   1:  PR[GP1:91,1] = PR[GP1:90,1] + 51.280;
   1:  PR[GP1:91,2] = PR[GP1:90,2] + -7.015;
   1:L PR[91] 10mm/sec CNT100;
   1:  PR[GP1:91,1] = PR[GP1:90,1] + 52.296;
   1:  PR[GP1:91,2] = PR[GP1:90,2] + 0.271;
   1:L PR[91] 10mm/sec CNT100;
   1:  PR[GP1:91,1] = PR[GP1:90,1] + 51.315;
   1:  PR[GP1:91,2] = PR[GP1:90,2] + 6.204;
   1:L PR[91] 10mm/sec CNT100;
   1:  PR[GP1:91,1] = PR[GP1:90,1] + 50.273;
   1:  PR[GP1:91,2] = PR[GP1:90,2] + 13.672;
   1:L PR[91] 10mm/sec CNT100;
   1:  PR[GP1:91,1] = PR[GP1:90,1] + 47.241;
   1:  PR[GP1:91,2] = PR[GP1:90,2] + 20.539;
   1:L PR[91] 10mm/sec CNT100;
   1:  PR[GP1:91,1] = PR[GP1:90,1] + 44.357;
   1:  PR[GP1:91,2] = PR[GP1:90,2] + 25.832;
   1:L PR[91] 10mm/sec CNT100;
   1:  PR[GP1:91,1] = PR[GP1:90,1] + 39.468;
   1:  PR[GP1:91,2] = PR[GP1:90,2] + 31.722;
   1:L PR[91] 10mm/sec CNT100;
   1:  PR[GP1:91,1] = PR[GP1:90,1] + 35.135;
   1:  PR[GP1:91,2] = PR[GP1:90,2] + 35.737;
   1:L PR[91] 10mm/sec CNT100;
   1:  PR[GP1:91,1] = PR[GP1:90,1] + 26.217;
   1:  PR[GP1:91,2] = PR[GP1:90,2] + 41.260;
   1:L PR[91] 10mm/sec CNT100;
   1:  PR[GP1:91,1] = PR[GP1:90,1] + 20.960;
   1:  PR[GP1:91,2] = PR[GP1:90,2] + 43.644;
   1:L PR[91] 10mm/sec CNT100;
   1:  PR[GP1:91,1] = PR[GP1:90,1] + 10.344;
   1:  PR[GP1:91,2] = PR[GP1:90,2] + 45.629;
   1:L PR[91] 10mm/sec CNT100;
   1:  PR[GP1:91,1] = PR[GP1:90,1] + 4.776;
   1:  PR[GP1:91,2] = PR[GP1:90,2] + 46.223;
   1:L PR[91] 10mm/sec CNT100;
   1:  PR[GP1:91,1] = PR[GP1:90,1] + -0.263;
   1:  PR[GP1:91,2] = PR[GP1:90,2] + 45.337;
   1:L PR[91] 10mm/sec CNT100;
   1:  PR[GP1:91,1] = PR[GP1:90,1] + -5.307;
   1:  PR[GP1:91,2] = PR[GP1:90,2] + 46.223;
   1:L PR[91] 10mm/sec CNT100;
   1:  PR[GP1:91,1] = PR[GP1:90,1] + -10.875;
   1:  PR[GP1:91,2] = PR[GP1:90,2] + 45.629;
   1:L PR[91] 10mm/sec CNT100;
   1:  PR[GP1:91,1] = PR[GP1:90,1] + -21.488;
   1:  PR[GP1:91,2] = PR[GP1:90,2] + 43.644;
   1:L PR[91] 10mm/sec CNT100;
   1:  PR[GP1:91,1] = PR[GP1:90,1] + -26.745;
   1:  PR[GP1:91,2] = PR[GP1:90,2] + 41.258;
   1:L PR[91] 10mm/sec CNT100;
   1:  PR[GP1:91,1] = PR[GP1:90,1] + -35.660;
   1:  PR[GP1:91,2] = PR[GP1:90,2] + 35.736;
   1:L PR[91] 10mm/sec CNT100;
   1:  PR[GP1:91,1] = PR[GP1:90,1] + -39.993;
   1:  PR[GP1:91,2] = PR[GP1:90,2] + 31.727;
   1:L PR[91] 10mm/sec CNT100;
   1:  PR[GP1:91,1] = PR[GP1:90,1] + -44.883;
   1:  PR[GP1:91,2] = PR[GP1:90,2] + 25.837;
   1:L PR[91] 10mm/sec CNT100;
   1:  PR[GP1:91,1] = PR[GP1:90,1] + -47.767;
   1:  PR[GP1:91,2] = PR[GP1:90,2] + 20.534;
   1:L PR[91] 10mm/sec CNT100;
   1:  PR[GP1:91,1] = PR[GP1:90,1] + -50.803;
   1:  PR[GP1:91,2] = PR[GP1:90,2] + 13.658;
   1:L PR[91] 10mm/sec CNT100;
   1:  PR[GP1:91,1] = PR[GP1:90,1] + -51.805;
   1:  PR[GP1:91,2] = PR[GP1:90,2] + 7.716;
   1:L PR[91] 10mm/sec CNT100;
   1:  PR[GP1:91,1] = PR[GP1:90,1] + -51.806;
   1:  PR[GP1:91,2] = PR[GP1:90,2] + 7.573;
   1:L PR[91] 10mm/sec CNT100;
   1:  PR[GP1:91,1] = PR[GP1:90,1] + -52.823;
   1:  PR[GP1:91,2] = PR[GP1:90,2] + 0.287;
   1:L PR[91] 10mm/sec CNT100;
   1:  PR[GP1:91,1] = PR[GP1:90,1] + -51.845;
   1:  PR[GP1:91,2] = PR[GP1:90,2] + -5.627;
   1:L PR[91] 10mm/sec CNT100;
   1:  PR[GP1:91,1] = PR[GP1:90,1] + -50.804;
   1:  PR[GP1:91,2] = PR[GP1:90,2] + -13.095;
   1:L PR[91] 10mm/sec CNT100;
   1:  PR[GP1:91,1] = PR[GP1:90,1] + -47.772;
   1:  PR[GP1:91,2] = PR[GP1:90,2] + -19.963;
   1:L PR[91] 10mm/sec CNT100;
   1:  PR[GP1:91,1] = PR[GP1:90,1] + -44.899;
   1:  PR[GP1:91,2] = PR[GP1:90,2] + -25.258;
   1:L PR[91] 10mm/sec CNT100;
   1:  PR[GP1:91,1] = PR[GP1:90,1] + -40.009;
   1:  PR[GP1:91,2] = PR[GP1:90,2] + -31.148;
   1:L PR[91] 10mm/sec CNT100;
   1:  PR[GP1:91,1] = PR[GP1:90,1] + -35.691;
   1:  PR[GP1:91,2] = PR[GP1:90,2] + -35.157;
   1:L PR[91] 10mm/sec CNT100;
   1:  PR[GP1:91,1] = PR[GP1:90,1] + -26.777;
   1:  PR[GP1:91,2] = PR[GP1:90,2] + -40.678;
   1:L PR[91] 10mm/sec CNT100;
   1:  PR[GP1:91,1] = PR[GP1:90,1] + -21.535;
   1:  PR[GP1:91,2] = PR[GP1:90,2] + -43.073;
   1:L PR[91] 10mm/sec CNT100;
   1:  PR[GP1:91,1] = PR[GP1:90,1] + -10.924;
   1:  PR[GP1:91,2] = PR[GP1:90,2] + -45.058;
   1:L PR[91] 10mm/sec CNT100;
   1:  PR[GP1:91,1] = PR[GP1:90,1] + -5.362;
   1:  PR[GP1:91,2] = PR[GP1:90,2] + -45.668;
   1:L PR[91] 10mm/sec CNT100;
   1:  PR[GP1:91,1] = PR[GP1:90,1] + -0.263;
   1:  PR[GP1:91,2] = PR[GP1:90,2] + -44.813;
   1:L PR[91] 10mm/sec CNT100;
   1:  PR[GP1:91,1] = PR[GP1:90,1] + 4.642;
   1:  PR[GP1:91,2] = PR[GP1:90,2] + -45.797;
   1:  PR[GP1:91,3] = PR[GP1:90,3] + 112.545;
   1:L PR[91] 10mm/sec CNT100;
   1:  PR[GP1:91,1] = PR[GP1:90,1] + 9.992;
   1:  PR[GP1:91,2] = PR[GP1:90,2] + -45.209;
   1:L PR[91] 10mm/sec CNT100;
   1:  PR[GP1:91,1] = PR[GP1:90,1] + 20.880;
   1:  PR[GP1:91,2] = PR[GP1:90,2] + -43.174;
   1:L PR[91] 10mm/sec CNT100;
   1:  PR[GP1:91,1] = PR[GP1:90,1] + 25.924;
   1:  PR[GP1:91,2] = PR[GP1:90,2] + -40.872;
   1:L PR[91] 10mm/sec CNT100;
   1:  PR[GP1:91,1] = PR[GP1:90,1] + 35.087;
   1:  PR[GP1:91,2] = PR[GP1:90,2] + -35.196;
   1:L PR[91] 10mm/sec CNT100;
   1:  PR[GP1:91,1] = PR[GP1:90,1] + 39.242;
   1:  PR[GP1:91,2] = PR[GP1:90,2] + -31.334;
   1:L PR[91] 10mm/sec CNT100;
   1:  PR[GP1:91,1] = PR[GP1:90,1] + 44.275;
   1:  PR[GP1:91,2] = PR[GP1:90,2] + -25.271;
   1:L PR[91] 10mm/sec CNT100;
   1:  PR[GP1:91,1] = PR[GP1:90,1] + 47.039;
   1:  PR[GP1:91,2] = PR[GP1:90,2] + -20.185;
   1:L PR[91] 10mm/sec CNT100;
   1:  PR[GP1:91,1] = PR[GP1:90,1] + 50.168;
   1:  PR[GP1:91,2] = PR[GP1:90,2] + -13.099;
   1:L PR[91] 10mm/sec CNT100;
   1:  PR[GP1:91,1] = PR[GP1:90,1] + 51.128;
   1:  PR[GP1:91,2] = PR[GP1:90,2] + -7.389;
   1:L PR[91] 10mm/sec CNT100;
   1:  PR[GP1:91,1] = PR[GP1:90,1] + 51.129;
   1:  PR[GP1:91,2] = PR[GP1:90,2] + -7.251;
   1:L PR[91] 10mm/sec CNT100;
   1:  PR[GP1:91,1] = PR[GP1:90,1] + 52.178;
   1:  PR[GP1:91,2] = PR[GP1:90,2] + 0.271;
   1:L PR[91] 10mm/sec CNT100;
   1:  PR[GP1:91,1] = PR[GP1:90,1] + 51.234;
   1:  PR[GP1:91,2] = PR[GP1:90,2] + 5.979;
   1:L PR[91] 10mm/sec CNT100;
   1:  PR[GP1:91,1] = PR[GP1:90,1] + 50.160;
   1:  PR[GP1:91,2] = PR[GP1:90,2] + 13.676;
   1:L PR[91] 10mm/sec CNT100;
   1:  PR[GP1:91,1] = PR[GP1:90,1] + 47.035;
   1:  PR[GP1:91,2] = PR[GP1:90,2] + 20.755;
   1:L PR[91] 10mm/sec CNT100;
   1:  PR[GP1:91,1] = PR[GP1:90,1] + 44.260;
   1:  PR[GP1:91,2] = PR[GP1:90,2] + 25.848;
   1:L PR[91] 10mm/sec CNT100;
   1:  PR[GP1:91,1] = PR[GP1:90,1] + 39.227;
   1:  PR[GP1:91,2] = PR[GP1:90,2] + 31.912;
   1:L PR[91] 10mm/sec CNT100;
   1:  PR[GP1:91,1] = PR[GP1:90,1] + 35.058;
   1:  PR[GP1:91,2] = PR[GP1:90,2] + 35.774;
   1:L PR[91] 10mm/sec CNT100;
   1:  PR[GP1:91,1] = PR[GP1:90,1] + 25.893;
   1:  PR[GP1:91,2] = PR[GP1:90,2] + 41.450;
   1:L PR[91] 10mm/sec CNT100;
   1:  PR[GP1:91,1] = PR[GP1:90,1] + 20.836;
   1:  PR[GP1:91,2] = PR[GP1:90,2] + 43.744;
   1:L PR[91] 10mm/sec CNT100;
   1:  PR[GP1:91,1] = PR[GP1:90,1] + 9.945;
   1:  PR[GP1:91,2] = PR[GP1:90,2] + 45.780;
   1:L PR[91] 10mm/sec CNT100;
   1:  PR[GP1:91,1] = PR[GP1:90,1] + 4.588;
   1:  PR[GP1:91,2] = PR[GP1:90,2] + 46.352;
   1:L PR[91] 10mm/sec CNT100;
   1:  PR[GP1:91,1] = PR[GP1:90,1] + -0.263;
   1:  PR[GP1:91,2] = PR[GP1:90,2] + 45.499;
   1:L PR[91] 10mm/sec CNT100;
   1:  PR[GP1:91,1] = PR[GP1:90,1] + -5.120;
   1:  PR[GP1:91,2] = PR[GP1:90,2] + 46.352;
   1:L PR[91] 10mm/sec CNT100;
   1:  PR[GP1:91,1] = PR[GP1:90,1] + -10.477;
   1:  PR[GP1:91,2] = PR[GP1:90,2] + 45.780;
   1:L PR[91] 10mm/sec CNT100;
   1:  PR[GP1:91,1] = PR[GP1:90,1] + -21.364;
   1:  PR[GP1:91,2] = PR[GP1:90,2] + 43.744;
   1:L PR[91] 10mm/sec CNT100;
   1:  PR[GP1:91,1] = PR[GP1:90,1] + -26.421;
   1:  PR[GP1:91,2] = PR[GP1:90,2] + 41.448;
   1:L PR[91] 10mm/sec CNT100;
   1:  PR[GP1:91,1] = PR[GP1:90,1] + -35.583;
   1:  PR[GP1:91,2] = PR[GP1:90,2] + 35.774;
   1:L PR[91] 10mm/sec CNT100;
   1:  PR[GP1:91,1] = PR[GP1:90,1] + -39.752;
   1:  PR[GP1:91,2] = PR[GP1:90,2] + 31.916;
   1:L PR[91] 10mm/sec CNT100;
   1:  PR[GP1:91,1] = PR[GP1:90,1] + -44.786;
   1:  PR[GP1:91,2] = PR[GP1:90,2] + 25.852;
   1:L PR[91] 10mm/sec CNT100;
   1:  PR[GP1:91,1] = PR[GP1:90,1] + -47.561;
   1:  PR[GP1:91,2] = PR[GP1:90,2] + 20.750;
   1:L PR[91] 10mm/sec CNT100;
   1:  PR[GP1:91,1] = PR[GP1:90,1] + -50.690;
   1:  PR[GP1:91,2] = PR[GP1:90,2] + 13.662;
   1:L PR[91] 10mm/sec CNT100;
   1:  PR[GP1:91,1] = PR[GP1:90,1] + -51.654;
   1:  PR[GP1:91,2] = PR[GP1:90,2] + 7.947;
   1:L PR[91] 10mm/sec CNT100;
   1:  PR[GP1:91,1] = PR[GP1:90,1] + -51.655;
   1:  PR[GP1:91,2] = PR[GP1:90,2] + 7.809;
   1:L PR[91] 10mm/sec CNT100;
   1:  PR[GP1:91,1] = PR[GP1:90,1] + -52.705;
   1:  PR[GP1:91,2] = PR[GP1:90,2] + 0.287;
   1:L PR[91] 10mm/sec CNT100;
   1:  PR[GP1:91,1] = PR[GP1:90,1] + -51.764;
   1:  PR[GP1:91,2] = PR[GP1:90,2] + -5.404;
   1:L PR[91] 10mm/sec CNT100;
   1:  PR[GP1:91,1] = PR[GP1:90,1] + -50.691;
   1:  PR[GP1:91,2] = PR[GP1:90,2] + -13.100;
   1:L PR[91] 10mm/sec CNT100;
   1:  PR[GP1:91,1] = PR[GP1:90,1] + -47.565;
   1:  PR[GP1:91,2] = PR[GP1:90,2] + -20.180;
   1:L PR[91] 10mm/sec CNT100;
   1:  PR[GP1:91,1] = PR[GP1:90,1] + -44.801;
   1:  PR[GP1:91,2] = PR[GP1:90,2] + -25.275;
   1:L PR[91] 10mm/sec CNT100;
   1:  PR[GP1:91,1] = PR[GP1:90,1] + -39.767;
   1:  PR[GP1:91,2] = PR[GP1:90,2] + -31.338;
   1:L PR[91] 10mm/sec CNT100;
   1:  PR[GP1:91,1] = PR[GP1:90,1] + -35.613;
   1:  PR[GP1:91,2] = PR[GP1:90,2] + -35.196;
   1:L PR[91] 10mm/sec CNT100;
   1:  PR[GP1:91,1] = PR[GP1:90,1] + -26.452;
   1:  PR[GP1:91,2] = PR[GP1:90,2] + -40.870;
   1:L PR[91] 10mm/sec CNT100;
   1:  PR[GP1:91,1] = PR[GP1:90,1] + -21.409;
   1:  PR[GP1:91,2] = PR[GP1:90,2] + -43.174;
   1:L PR[91] 10mm/sec CNT100;
   1:  PR[GP1:91,1] = PR[GP1:90,1] + -10.524;
   1:  PR[GP1:91,2] = PR[GP1:90,2] + -45.210;
   1:L PR[91] 10mm/sec CNT100;
   1:  PR[GP1:91,1] = PR[GP1:90,1] + -5.173;
   1:  PR[GP1:91,2] = PR[GP1:90,2] + -45.797;
   1:L PR[91] 10mm/sec CNT100;
   1:  PR[GP1:91,1] = PR[GP1:90,1] + -0.263;
   1:  PR[GP1:91,2] = PR[GP1:90,2] + -44.973;
   1:L PR[91] 10mm/sec CNT100;
   1:  PR[GP1:91,1] = PR[GP1:90,1] + 4.452;
   1:  PR[GP1:91,2] = PR[GP1:90,2] + -45.925;
   1:  PR[GP1:91,3] = PR[GP1:90,3] + 113.155;
   1:L PR[91] 10mm/sec CNT100;
   1:  PR[GP1:91,1] = PR[GP1:90,1] + 9.591;
   1:  PR[GP1:91,2] = PR[GP1:90,2] + -45.361;
   1:L PR[91] 10mm/sec CNT100;
   1:  PR[GP1:91,1] = PR[GP1:90,1] + 20.754;
   1:  PR[GP1:91,2] = PR[GP1:90,2] + -43.274;
   1:L PR[91] 10mm/sec CNT100;
   1:  PR[GP1:91,1] = PR[GP1:90,1] + 25.598;
   1:  PR[GP1:91,2] = PR[GP1:90,2] + -41.063;
   1:L PR[91] 10mm/sec CNT100;
   1:  PR[GP1:91,1] = PR[GP1:90,1] + 35.009;
   1:  PR[GP1:91,2] = PR[GP1:90,2] + -35.235;
   1:L PR[91] 10mm/sec CNT100;
   1:  PR[GP1:91,1] = PR[GP1:90,1] + 39.000;
   1:  PR[GP1:91,2] = PR[GP1:90,2] + -31.525;
   1:L PR[91] 10mm/sec CNT100;
   1:  PR[GP1:91,1] = PR[GP1:90,1] + 44.178;
   1:  PR[GP1:91,2] = PR[GP1:90,2] + -25.287;
   1:L PR[91] 10mm/sec CNT100;
   1:  PR[GP1:91,1] = PR[GP1:90,1] + 46.833;
   1:  PR[GP1:91,2] = PR[GP1:90,2] + -20.402;
   1:L PR[91] 10mm/sec CNT100;
   1:  PR[GP1:91,1] = PR[GP1:90,1] + 50.055;
   1:  PR[GP1:91,2] = PR[GP1:90,2] + -13.104;
   1:L PR[91] 10mm/sec CNT100;
   1:  PR[GP1:91,1] = PR[GP1:90,1] + 50.977;
   1:  PR[GP1:91,2] = PR[GP1:90,2] + -7.619;
   1:L PR[91] 10mm/sec CNT100;
   1:  PR[GP1:91,1] = PR[GP1:90,1] + 50.978;
   1:  PR[GP1:91,2] = PR[GP1:90,2] + -7.487;
   1:L PR[91] 10mm/sec CNT100;
   1:  PR[GP1:91,1] = PR[GP1:90,1] + 52.060;
   1:  PR[GP1:91,2] = PR[GP1:90,2] + 0.271;
   1:L PR[91] 10mm/sec CNT100;
   1:  PR[GP1:91,1] = PR[GP1:90,1] + 51.153;
   1:  PR[GP1:91,2] = PR[GP1:90,2] + 5.755;
   1:L PR[91] 10mm/sec CNT100;
   1:  PR[GP1:91,1] = PR[GP1:90,1] + 50.048;
   1:  PR[GP1:91,2] = PR[GP1:90,2] + 13.681;
   1:L PR[91] 10mm/sec CNT100;
   1:  PR[GP1:91,1] = PR[GP1:90,1] + 46.829;
   1:  PR[GP1:91,2] = PR[GP1:90,2] + 20.971;
   1:L PR[91] 10mm/sec CNT100;
   1:  PR[GP1:91,1] = PR[GP1:90,1] + 44.163;
   1:  PR[GP1:91,2] = PR[GP1:90,2] + 25.864;
   1:L PR[91] 10mm/sec CNT100;
   1:  PR[GP1:91,1] = PR[GP1:90,1] + 38.985;
   1:  PR[GP1:91,2] = PR[GP1:90,2] + 32.102;
   1:L PR[91] 10mm/sec CNT100;
   1:  PR[GP1:91,1] = PR[GP1:90,1] + 34.980;
   1:  PR[GP1:91,2] = PR[GP1:90,2] + 35.812;
   1:L PR[91] 10mm/sec CNT100;
   1:  PR[GP1:91,1] = PR[GP1:90,1] + 25.569;
   1:  PR[GP1:91,2] = PR[GP1:90,2] + 41.641;
   1:L PR[91] 10mm/sec CNT100;
   1:  PR[GP1:91,1] = PR[GP1:90,1] + 20.711;
   1:  PR[GP1:91,2] = PR[GP1:90,2] + 43.844;
   1:L PR[91] 10mm/sec CNT100;
   1:  PR[GP1:91,1] = PR[GP1:90,1] + 9.547;
   1:  PR[GP1:91,2] = PR[GP1:90,2] + 45.931;
   1:L PR[91] 10mm/sec CNT100;
   1:  PR[GP1:91,1] = PR[GP1:90,1] + 4.401;
   1:  PR[GP1:91,2] = PR[GP1:90,2] + 46.480;
   1:L PR[91] 10mm/sec CNT100;
   1:  PR[GP1:91,1] = PR[GP1:90,1] + -0.263;
   1:  PR[GP1:91,2] = PR[GP1:90,2] + 45.660;
   1:L PR[91] 10mm/sec CNT100;
   1:  PR[GP1:91,1] = PR[GP1:90,1] + -4.933;
   1:  PR[GP1:91,2] = PR[GP1:90,2] + 46.480;
   1:L PR[91] 10mm/sec CNT100;
   1:  PR[GP1:91,1] = PR[GP1:90,1] + -10.078;
   1:  PR[GP1:91,2] = PR[GP1:90,2] + 45.931;
   1:L PR[91] 10mm/sec CNT100;
   1:  PR[GP1:91,1] = PR[GP1:90,1] + -21.240;
   1:  PR[GP1:91,2] = PR[GP1:90,2] + 43.844;
   1:L PR[91] 10mm/sec CNT100;
   1:  PR[GP1:91,1] = PR[GP1:90,1] + -26.097;
   1:  PR[GP1:91,2] = PR[GP1:90,2] + 41.639;
   1:L PR[91] 10mm/sec CNT100;
   1:  PR[GP1:91,1] = PR[GP1:90,1] + -35.506;
   1:  PR[GP1:91,2] = PR[GP1:90,2] + 35.811;
   1:L PR[91] 10mm/sec CNT100;
   1:  PR[GP1:91,1] = PR[GP1:90,1] + -39.511;
   1:  PR[GP1:91,2] = PR[GP1:90,2] + 32.106;
   1:L PR[91] 10mm/sec CNT100;
   1:  PR[GP1:91,1] = PR[GP1:90,1] + -44.689;
   1:  PR[GP1:91,2] = PR[GP1:90,2] + 25.868;
   1:L PR[91] 10mm/sec CNT100;
   1:  PR[GP1:91,1] = PR[GP1:90,1] + -47.355;
   1:  PR[GP1:91,2] = PR[GP1:90,2] + 20.966;
   1:L PR[91] 10mm/sec CNT100;
   1:  PR[GP1:91,1] = PR[GP1:90,1] + -50.577;
   1:  PR[GP1:91,2] = PR[GP1:90,2] + 13.667;
   1:L PR[91] 10mm/sec CNT100;
   1:  PR[GP1:91,1] = PR[GP1:90,1] + -51.503;
   1:  PR[GP1:91,2] = PR[GP1:90,2] + 8.177;
   1:L PR[91] 10mm/sec CNT100;
   1:  PR[GP1:91,1] = PR[GP1:90,1] + -51.504;
   1:  PR[GP1:91,2] = PR[GP1:90,2] + 8.046;
   1:L PR[91] 10mm/sec CNT100;
   1:  PR[GP1:91,1] = PR[GP1:90,1] + -52.587;
   1:  PR[GP1:91,2] = PR[GP1:90,2] + 0.287;
   1:L PR[91] 10mm/sec CNT100;
   1:  PR[GP1:91,1] = PR[GP1:90,1] + -51.683;
   1:  PR[GP1:91,2] = PR[GP1:90,2] + -5.180;
   1:L PR[91] 10mm/sec CNT100;
   1:  PR[GP1:91,1] = PR[GP1:90,1] + -50.578;
   1:  PR[GP1:91,2] = PR[GP1:90,2] + -13.106;
   1:L PR[91] 10mm/sec CNT100;
   1:  PR[GP1:91,1] = PR[GP1:90,1] + -47.359;
   1:  PR[GP1:91,2] = PR[GP1:90,2] + -20.396;
   1:L PR[91] 10mm/sec CNT100;
   1:  PR[GP1:91,1] = PR[GP1:90,1] + -44.704;
   1:  PR[GP1:91,2] = PR[GP1:90,2] + -25.291;
   1:L PR[91] 10mm/sec CNT100;
   1:  PR[GP1:91,1] = PR[GP1:90,1] + -39.525;
   1:  PR[GP1:91,2] = PR[GP1:90,2] + -31.529;
   1:L PR[91] 10mm/sec CNT100;
   1:  PR[GP1:91,1] = PR[GP1:90,1] + -35.535;
   1:  PR[GP1:91,2] = PR[GP1:90,2] + -35.234;
   1:L PR[91] 10mm/sec CNT100;
   1:  PR[GP1:91,1] = PR[GP1:90,1] + -26.127;
   1:  PR[GP1:91,2] = PR[GP1:90,2] + -41.061;
   1:L PR[91] 10mm/sec CNT100;
   1:  PR[GP1:91,1] = PR[GP1:90,1] + -21.282;
   1:  PR[GP1:91,2] = PR[GP1:90,2] + -43.274;
   1:L PR[91] 10mm/sec CNT100;
   1:  PR[GP1:91,1] = PR[GP1:90,1] + -10.123;
   1:  PR[GP1:91,2] = PR[GP1:90,2] + -45.361;
   1:L PR[91] 10mm/sec CNT100;
   1:  PR[GP1:91,1] = PR[GP1:90,1] + -4.984;
   1:  PR[GP1:91,2] = PR[GP1:90,2] + -45.925;
   1:L PR[91] 10mm/sec CNT100;
   1:  PR[GP1:91,1] = PR[GP1:90,1] + -0.263;
   1:  PR[GP1:91,2] = PR[GP1:90,2] + -45.134;
   1:L PR[91] 10mm/sec CNT100;
   1:  PR[GP1:91,1] = PR[GP1:90,1] + 4.263;
   1:  PR[GP1:91,2] = PR[GP1:90,2] + -46.054;
   1:  PR[GP1:91,3] = PR[GP1:90,3] + 113.765;
   1:L PR[91] 10mm/sec CNT100;
   1:  PR[GP1:91,1] = PR[GP1:90,1] + 9.191;
   1:  PR[GP1:91,2] = PR[GP1:90,2] + -45.512;
   1:L PR[91] 10mm/sec CNT100;
   1:  PR[GP1:91,1] = PR[GP1:90,1] + 20.628;
   1:  PR[GP1:91,2] = PR[GP1:90,2] + -43.375;
   1:L PR[91] 10mm/sec CNT100;
   1:  PR[GP1:91,1] = PR[GP1:90,1] + 25.273;
   1:  PR[GP1:91,2] = PR[GP1:90,2] + -41.254;
   1:L PR[91] 10mm/sec CNT100;
   1:  PR[GP1:91,1] = PR[GP1:90,1] + 34.931;
   1:  PR[GP1:91,2] = PR[GP1:90,2] + -35.273;
   1:L PR[91] 10mm/sec CNT100;
   1:  PR[GP1:91,1] = PR[GP1:90,1] + 38.758;
   1:  PR[GP1:91,2] = PR[GP1:90,2] + -31.715;
   1:L PR[91] 10mm/sec CNT100;
   1:  PR[GP1:91,1] = PR[GP1:90,1] + 44.080;
   1:  PR[GP1:91,2] = PR[GP1:90,2] + -25.304;
   1:L PR[91] 10mm/sec CNT100;
   1:  PR[GP1:91,1] = PR[GP1:90,1] + 46.627;
   1:  PR[GP1:91,2] = PR[GP1:90,2] + -20.618;
   1:L PR[91] 10mm/sec CNT100;
   1:  PR[GP1:91,1] = PR[GP1:90,1] + 49.942;
   1:  PR[GP1:91,2] = PR[GP1:90,2] + -13.109;
   1:L PR[91] 10mm/sec CNT100;
   1:  PR[GP1:91,1] = PR[GP1:90,1] + 50.826;
   1:  PR[GP1:91,2] = PR[GP1:90,2] + -7.850;
   1:L PR[91] 10mm/sec CNT100;
   1:  PR[GP1:91,1] = PR[GP1:90,1] + 50.827;
   1:  PR[GP1:91,2] = PR[GP1:90,2] + -7.724;
   1:L PR[91] 10mm/sec CNT100;
   1:  PR[GP1:91,1] = PR[GP1:90,1] + 51.942;
   1:  PR[GP1:91,2] = PR[GP1:90,2] + 0.271;
   1:L PR[91] 10mm/sec CNT100;
   1:  PR[GP1:91,1] = PR[GP1:90,1] + 51.072;
   1:  PR[GP1:91,2] = PR[GP1:90,2] + 5.531;
   1:L PR[91] 10mm/sec CNT100;
   1:  PR[GP1:91,1] = PR[GP1:90,1] + 49.935;
   1:  PR[GP1:91,2] = PR[GP1:90,2] + 13.685;
   1:L PR[91] 10mm/sec CNT100;
   1:  PR[GP1:91,1] = PR[GP1:90,1] + 46.623;
   1:  PR[GP1:91,2] = PR[GP1:90,2] + 21.187;
   1:L PR[91] 10mm/sec CNT100;
   1:  PR[GP1:91,1] = PR[GP1:90,1] + 44.066;
   1:  PR[GP1:91,2] = PR[GP1:90,2] + 25.880;
   1:L PR[91] 10mm/sec CNT100;
   1:  PR[GP1:91,1] = PR[GP1:90,1] + 38.744;
   1:  PR[GP1:91,2] = PR[GP1:90,2] + 32.291;
   1:L PR[91] 10mm/sec CNT100;
   1:  PR[GP1:91,1] = PR[GP1:90,1] + 34.903;
   1:  PR[GP1:91,2] = PR[GP1:90,2] + 35.849;
   1:L PR[91] 10mm/sec CNT100;
   1:  PR[GP1:91,1] = PR[GP1:90,1] + 25.244;
   1:  PR[GP1:91,2] = PR[GP1:90,2] + 41.831;
   1:L PR[91] 10mm/sec CNT100;
   1:  PR[GP1:91,1] = PR[GP1:90,1] + 20.587;
   1:  PR[GP1:91,2] = PR[GP1:90,2] + 43.944;
   1:L PR[91] 10mm/sec CNT100;
   1:  PR[GP1:91,1] = PR[GP1:90,1] + 9.148;
   1:  PR[GP1:91,2] = PR[GP1:90,2] + 46.082;
   1:L PR[91] 10mm/sec CNT100;
   1:  PR[GP1:91,1] = PR[GP1:90,1] + 4.214;
   1:  PR[GP1:91,2] = PR[GP1:90,2] + 46.609;
   1:L PR[91] 10mm/sec CNT100;
   1:  PR[GP1:91,1] = PR[GP1:90,1] + -0.263;
   1:  PR[GP1:91,2] = PR[GP1:90,2] + 45.821;
   1:L PR[91] 10mm/sec CNT100;
   1:  PR[GP1:91,1] = PR[GP1:90,1] + -4.746;
   1:  PR[GP1:91,2] = PR[GP1:90,2] + 46.609;
   1:L PR[91] 10mm/sec CNT100;
   1:  PR[GP1:91,1] = PR[GP1:90,1] + -9.679;
   1:  PR[GP1:91,2] = PR[GP1:90,2] + 46.082;
   1:L PR[91] 10mm/sec CNT100;
   1:  PR[GP1:91,1] = PR[GP1:90,1] + -21.115;
   1:  PR[GP1:91,2] = PR[GP1:90,2] + 43.944;
   1:L PR[91] 10mm/sec CNT100;
   1:  PR[GP1:91,1] = PR[GP1:90,1] + -25.772;
   1:  PR[GP1:91,2] = PR[GP1:90,2] + 41.829;
   1:L PR[91] 10mm/sec CNT100;
   1:  PR[GP1:91,1] = PR[GP1:90,1] + -35.429;
   1:  PR[GP1:91,2] = PR[GP1:90,2] + 35.849;
   1:L PR[91] 10mm/sec CNT100;
   1:  PR[GP1:91,1] = PR[GP1:90,1] + -39.269;
   1:  PR[GP1:91,2] = PR[GP1:90,2] + 32.295;
   1:L PR[91] 10mm/sec CNT100;
   1:  PR[GP1:91,1] = PR[GP1:90,1] + -44.592;
   1:  PR[GP1:91,2] = PR[GP1:90,2] + 25.884;
   1:L PR[91] 10mm/sec CNT100;
   1:  PR[GP1:91,1] = PR[GP1:90,1] + -47.149;
   1:  PR[GP1:91,2] = PR[GP1:90,2] + 21.182;
   1:L PR[91] 10mm/sec CNT100;
   1:  PR[GP1:91,1] = PR[GP1:90,1] + -50.465;
   1:  PR[GP1:91,2] = PR[GP1:90,2] + 13.672;
   1:L PR[91] 10mm/sec CNT100;
   1:  PR[GP1:91,1] = PR[GP1:90,1] + -51.352;
   1:  PR[GP1:91,2] = PR[GP1:90,2] + 8.408;
   1:L PR[91] 10mm/sec CNT100;
   1:  PR[GP1:91,1] = PR[GP1:90,1] + -51.353;
   1:  PR[GP1:91,2] = PR[GP1:90,2] + 8.282;
   1:L PR[91] 10mm/sec CNT100;
   1:  PR[GP1:91,1] = PR[GP1:90,1] + -52.469;
   1:  PR[GP1:91,2] = PR[GP1:90,2] + 0.287;
   1:L PR[91] 10mm/sec CNT100;
   1:  PR[GP1:91,1] = PR[GP1:90,1] + -51.602;
   1:  PR[GP1:91,2] = PR[GP1:90,2] + -4.957;
   1:L PR[91] 10mm/sec CNT100;
   1:  PR[GP1:91,1] = PR[GP1:90,1] + -50.465;
   1:  PR[GP1:91,2] = PR[GP1:90,2] + -13.111;
   1:L PR[91] 10mm/sec CNT100;
   1:  PR[GP1:91,1] = PR[GP1:90,1] + -47.153;
   1:  PR[GP1:91,2] = PR[GP1:90,2] + -20.613;
   1:L PR[91] 10mm/sec CNT100;
   1:  PR[GP1:91,1] = PR[GP1:90,1] + -44.606;
   1:  PR[GP1:91,2] = PR[GP1:90,2] + -25.308;
   1:L PR[91] 10mm/sec CNT100;
   1:  PR[GP1:91,1] = PR[GP1:90,1] + -39.283;
   1:  PR[GP1:91,2] = PR[GP1:90,2] + -31.719;
   1:L PR[91] 10mm/sec CNT100;
   1:  PR[GP1:91,1] = PR[GP1:90,1] + -35.456;
   1:  PR[GP1:91,2] = PR[GP1:90,2] + -35.272;
   1:L PR[91] 10mm/sec CNT100;
   1:  PR[GP1:91,1] = PR[GP1:90,1] + -25.801;
   1:  PR[GP1:91,2] = PR[GP1:90,2] + -41.252;
   1:L PR[91] 10mm/sec CNT100;
   1:  PR[GP1:91,1] = PR[GP1:90,1] + -21.156;
   1:  PR[GP1:91,2] = PR[GP1:90,2] + -43.374;
   1:L PR[91] 10mm/sec CNT100;
   1:  PR[GP1:91,1] = PR[GP1:90,1] + -9.723;
   1:  PR[GP1:91,2] = PR[GP1:90,2] + -45.513;
   1:L PR[91] 10mm/sec CNT100;
   1:  PR[GP1:91,1] = PR[GP1:90,1] + -4.795;
   1:  PR[GP1:91,2] = PR[GP1:90,2] + -46.054;
   1:L PR[91] 10mm/sec CNT100;
   1:  PR[GP1:91,1] = PR[GP1:90,1] + -0.263;
   1:  PR[GP1:91,2] = PR[GP1:90,2] + -45.294;
   1:L PR[91] 10mm/sec CNT100;
   1:  PR[GP1:91,1] = PR[GP1:90,1] + 4.074;
   1:  PR[GP1:91,2] = PR[GP1:90,2] + -46.182;
   1:  PR[GP1:91,3] = PR[GP1:90,3] + 114.375;
   1:L PR[91] 10mm/sec CNT100;
   1:  PR[GP1:91,1] = PR[GP1:90,1] + 8.790;
   1:  PR[GP1:91,2] = PR[GP1:90,2] + -45.664;
   1:L PR[91] 10mm/sec CNT100;
   1:  PR[GP1:91,1] = PR[GP1:90,1] + 20.502;
   1:  PR[GP1:91,2] = PR[GP1:90,2] + -43.475;
   1:L PR[91] 10mm/sec CNT100;
   1:  PR[GP1:91,1] = PR[GP1:90,1] + 24.948;
   1:  PR[GP1:91,2] = PR[GP1:90,2] + -41.446;
   1:L PR[91] 10mm/sec CNT100;
   1:  PR[GP1:91,1] = PR[GP1:90,1] + 34.852;
   1:  PR[GP1:91,2] = PR[GP1:90,2] + -35.311;
   1:L PR[91] 10mm/sec CNT100;
   1:  PR[GP1:91,1] = PR[GP1:90,1] + 38.516;
   1:  PR[GP1:91,2] = PR[GP1:90,2] + -31.905;
   1:L PR[91] 10mm/sec CNT100;
   1:  PR[GP1:91,1] = PR[GP1:90,1] + 43.982;
   1:  PR[GP1:91,2] = PR[GP1:90,2] + -25.321;
   1:L PR[91] 10mm/sec CNT100;
   1:  PR[GP1:91,1] = PR[GP1:90,1] + 46.421;
   1:  PR[GP1:91,2] = PR[GP1:90,2] + -20.834;
   1:L PR[91] 10mm/sec CNT100;
   1:  PR[GP1:91,1] = PR[GP1:90,1] + 49.829;
   1:  PR[GP1:91,2] = PR[GP1:90,2] + -13.114;
   1:L PR[91] 10mm/sec CNT100;
   1:  PR[GP1:91,1] = PR[GP1:90,1] + 50.675;
   1:  PR[GP1:91,2] = PR[GP1:90,2] + -8.081;
   1:L PR[91] 10mm/sec CNT100;
   1:  PR[GP1:91,1] = PR[GP1:90,1] + 50.676;
   1:  PR[GP1:91,2] = PR[GP1:90,2] + -7.960;
   1:L PR[91] 10mm/sec CNT100;
   1:  PR[GP1:91,1] = PR[GP1:90,1] + 51.824;
   1:  PR[GP1:91,2] = PR[GP1:90,2] + 0.271;
   1:L PR[91] 10mm/sec CNT100;
   1:  PR[GP1:91,1] = PR[GP1:90,1] + 50.991;
   1:  PR[GP1:91,2] = PR[GP1:90,2] + 5.307;
   1:L PR[91] 10mm/sec CNT100;
   1:  PR[GP1:91,1] = PR[GP1:90,1] + 49.822;
   1:  PR[GP1:91,2] = PR[GP1:90,2] + 13.690;
   1:L PR[91] 10mm/sec CNT100;
   1:  PR[GP1:91,1] = PR[GP1:90,1] + 46.417;
   1:  PR[GP1:91,2] = PR[GP1:90,2] + 21.403;
   1:L PR[91] 10mm/sec CNT100;
   1:  PR[GP1:91,1] = PR[GP1:90,1] + 43.969;
   1:  PR[GP1:91,2] = PR[GP1:90,2] + 25.896;
   1:L PR[91] 10mm/sec CNT100;
   1:  PR[GP1:91,1] = PR[GP1:90,1] + 38.503;
   1:  PR[GP1:91,2] = PR[GP1:90,2] + 32.481;
   1:L PR[91] 10mm/sec CNT100;
   1:  PR[GP1:91,1] = PR[GP1:90,1] + 34.826;
   1:  PR[GP1:91,2] = PR[GP1:90,2] + 35.887;
   1:L PR[91] 10mm/sec CNT100;
   1:  PR[GP1:91,1] = PR[GP1:90,1] + 24.920;
   1:  PR[GP1:91,2] = PR[GP1:90,2] + 42.022;
   1:L PR[91] 10mm/sec CNT100;
   1:  PR[GP1:91,1] = PR[GP1:90,1] + 20.462;
   1:  PR[GP1:91,2] = PR[GP1:90,2] + 44.044;
   1:L PR[91] 10mm/sec CNT100;
   1:  PR[GP1:91,1] = PR[GP1:90,1] + 8.749;
   1:  PR[GP1:91,2] = PR[GP1:90,2] + 46.233;
   1:L PR[91] 10mm/sec CNT100;
   1:  PR[GP1:91,1] = PR[GP1:90,1] + 4.027;
   1:  PR[GP1:91,2] = PR[GP1:90,2] + 46.737;
   1:L PR[91] 10mm/sec CNT100;
   1:  PR[GP1:91,1] = PR[GP1:90,1] + -0.263;
   1:  PR[GP1:91,2] = PR[GP1:90,2] + 45.983;
   1:L PR[91] 10mm/sec CNT100;
   1:  PR[GP1:91,1] = PR[GP1:90,1] + -4.559;
   1:  PR[GP1:91,2] = PR[GP1:90,2] + 46.737;
   1:L PR[91] 10mm/sec CNT100;
   1:  PR[GP1:91,1] = PR[GP1:90,1] + -9.281;
   1:  PR[GP1:91,2] = PR[GP1:90,2] + 46.234;
   1:L PR[91] 10mm/sec CNT100;
   1:  PR[GP1:91,1] = PR[GP1:90,1] + -20.991;
   1:  PR[GP1:91,2] = PR[GP1:90,2] + 44.043;
   1:L PR[91] 10mm/sec CNT100;
   1:  PR[GP1:91,1] = PR[GP1:90,1] + -25.448;
   1:  PR[GP1:91,2] = PR[GP1:90,2] + 42.020;
   1:L PR[91] 10mm/sec CNT100;
   1:  PR[GP1:91,1] = PR[GP1:90,1] + -35.352;
   1:  PR[GP1:91,2] = PR[GP1:90,2] + 35.886;
   1:L PR[91] 10mm/sec CNT100;
   1:  PR[GP1:91,1] = PR[GP1:90,1] + -39.028;
   1:  PR[GP1:91,2] = PR[GP1:90,2] + 32.485;
   1:L PR[91] 10mm/sec CNT100;
   1:  PR[GP1:91,1] = PR[GP1:90,1] + -44.495;
   1:  PR[GP1:91,2] = PR[GP1:90,2] + 25.899;
   1:L PR[91] 10mm/sec CNT100;
   1:  PR[GP1:91,1] = PR[GP1:90,1] + -46.943;
   1:  PR[GP1:91,2] = PR[GP1:90,2] + 21.398;
   1:L PR[91] 10mm/sec CNT100;
   1:  PR[GP1:91,1] = PR[GP1:90,1] + -50.352;
   1:  PR[GP1:91,2] = PR[GP1:90,2] + 13.677;
   1:L PR[91] 10mm/sec CNT100;
   1:  PR[GP1:91,1] = PR[GP1:90,1] + -51.201;
   1:  PR[GP1:91,2] = PR[GP1:90,2] + 8.639;
   1:L PR[91] 10mm/sec CNT100;
   1:  PR[GP1:91,1] = PR[GP1:90,1] + -51.203;
   1:  PR[GP1:91,2] = PR[GP1:90,2] + 8.518;
   1:L PR[91] 10mm/sec CNT100;
   1:  PR[GP1:91,1] = PR[GP1:90,1] + -52.351;
   1:  PR[GP1:91,2] = PR[GP1:90,2] + 0.287;
   1:L PR[91] 10mm/sec CNT100;
   1:  PR[GP1:91,1] = PR[GP1:90,1] + -51.521;
   1:  PR[GP1:91,2] = PR[GP1:90,2] + -4.733;
   1:L PR[91] 10mm/sec CNT100;
   1:  PR[GP1:91,1] = PR[GP1:90,1] + -50.352;
   1:  PR[GP1:91,2] = PR[GP1:90,2] + -13.116;
   1:L PR[91] 10mm/sec CNT100;
   1:  PR[GP1:91,1] = PR[GP1:90,1] + -46.947;
   1:  PR[GP1:91,2] = PR[GP1:90,2] + -20.830;
   1:L PR[91] 10mm/sec CNT100;
   1:  PR[GP1:91,1] = PR[GP1:90,1] + -44.508;
   1:  PR[GP1:91,2] = PR[GP1:90,2] + -25.324;
   1:L PR[91] 10mm/sec CNT100;
   1:  PR[GP1:91,1] = PR[GP1:90,1] + -39.042;
   1:  PR[GP1:91,2] = PR[GP1:90,2] + -31.909;
   1:L PR[91] 10mm/sec CNT100;
   1:  PR[GP1:91,1] = PR[GP1:90,1] + -35.378;
   1:  PR[GP1:91,2] = PR[GP1:90,2] + -35.311;
   1:L PR[91] 10mm/sec CNT100;
   1:  PR[GP1:91,1] = PR[GP1:90,1] + -25.476;
   1:  PR[GP1:91,2] = PR[GP1:90,2] + -41.444;
   1:L PR[91] 10mm/sec CNT100;
   1:  PR[GP1:91,1] = PR[GP1:90,1] + -21.030;
   1:  PR[GP1:91,2] = PR[GP1:90,2] + -43.475;
   1:L PR[91] 10mm/sec CNT100;
   1:  PR[GP1:91,1] = PR[GP1:90,1] + -9.322;
   1:  PR[GP1:91,2] = PR[GP1:90,2] + -45.664;
   1:L PR[91] 10mm/sec CNT100;
   1:  PR[GP1:91,1] = PR[GP1:90,1] + -4.605;
   1:  PR[GP1:91,2] = PR[GP1:90,2] + -46.182;
   1:L PR[91] 10mm/sec CNT100;
   1:  PR[GP1:91,1] = PR[GP1:90,1] + -0.263;
   1:  PR[GP1:91,2] = PR[GP1:90,2] + -45.454;
   1:L PR[91] 10mm/sec CNT100;
   1:  PR[GP1:91,1] = PR[GP1:90,1] + 3.884;
   1:  PR[GP1:91,2] = PR[GP1:90,2] + -46.311;
   1:  PR[GP1:91,3] = PR[GP1:90,3] + 114.985;
   1:L PR[91] 10mm/sec CNT100;
   1:  PR[GP1:91,1] = PR[GP1:90,1] + 8.390;
   1:  PR[GP1:91,2] = PR[GP1:90,2] + -45.816;
   1:L PR[91] 10mm/sec CNT100;
   1:  PR[GP1:91,1] = PR[GP1:90,1] + 20.375;
   1:  PR[GP1:91,2] = PR[GP1:90,2] + -43.575;
   1:L PR[91] 10mm/sec CNT100;
   1:  PR[GP1:91,1] = PR[GP1:90,1] + 24.622;
   1:  PR[GP1:91,2] = PR[GP1:90,2] + -41.637;
   1:L PR[91] 10mm/sec CNT100;
   1:  PR[GP1:91,1] = PR[GP1:90,1] + 34.774;
   1:  PR[GP1:91,2] = PR[GP1:90,2] + -35.350;
   1:L PR[91] 10mm/sec CNT100;
   1:  PR[GP1:91,1] = PR[GP1:90,1] + 38.274;
   1:  PR[GP1:91,2] = PR[GP1:90,2] + -32.096;
   1:L PR[91] 10mm/sec CNT100;
   1:  PR[GP1:91,1] = PR[GP1:90,1] + 43.885;
   1:  PR[GP1:91,2] = PR[GP1:90,2] + -25.337;
   1:L PR[91] 10mm/sec CNT100;
   1:  PR[GP1:91,1] = PR[GP1:90,1] + 46.215;
   1:  PR[GP1:91,2] = PR[GP1:90,2] + -21.050;
   1:L PR[91] 10mm/sec CNT100;
   1:  PR[GP1:91,1] = PR[GP1:90,1] + 49.716;
   1:  PR[GP1:91,2] = PR[GP1:90,2] + -13.119;
   1:L PR[91] 10mm/sec CNT100;
   1:  PR[GP1:91,1] = PR[GP1:90,1] + 50.524;
   1:  PR[GP1:91,2] = PR[GP1:90,2] + -8.311;
   1:L PR[91] 10mm/sec CNT100;
   1:  PR[GP1:91,1] = PR[GP1:90,1] + 50.525;
   1:  PR[GP1:91,2] = PR[GP1:90,2] + -8.196;
   1:L PR[91] 10mm/sec CNT100;
   1:  PR[GP1:91,1] = PR[GP1:90,1] + 51.706;
   1:  PR[GP1:91,2] = PR[GP1:90,2] + 0.271;
   1:L PR[91] 10mm/sec CNT100;
   1:  PR[GP1:91,1] = PR[GP1:90,1] + 50.910;
   1:  PR[GP1:91,2] = PR[GP1:90,2] + 5.083;
   1:L PR[91] 10mm/sec CNT100;
   1:  PR[GP1:91,1] = PR[GP1:90,1] + 49.709;
   1:  PR[GP1:91,2] = PR[GP1:90,2] + 13.694;
   1:L PR[91] 10mm/sec CNT100;
   1:  PR[GP1:91,1] = PR[GP1:90,1] + 46.211;
   1:  PR[GP1:91,2] = PR[GP1:90,2] + 21.618;
   1:L PR[91] 10mm/sec CNT100;
   1:  PR[GP1:91,1] = PR[GP1:90,1] + 43.872;
   1:  PR[GP1:91,2] = PR[GP1:90,2] + 25.912;
   1:L PR[91] 10mm/sec CNT100;
   1:  PR[GP1:91,1] = PR[GP1:90,1] + 38.261;
   1:  PR[GP1:91,2] = PR[GP1:90,2] + 32.670;
   1:L PR[91] 10mm/sec CNT100;
   1:  PR[GP1:91,1] = PR[GP1:90,1] + 34.749;
   1:  PR[GP1:91,2] = PR[GP1:90,2] + 35.924;
   1:L PR[91] 10mm/sec CNT100;
   1:  PR[GP1:91,1] = PR[GP1:90,1] + 24.596;
   1:  PR[GP1:91,2] = PR[GP1:90,2] + 42.212;
   1:L PR[91] 10mm/sec CNT100;
   1:  PR[GP1:91,1] = PR[GP1:90,1] + 20.338;
   1:  PR[GP1:91,2] = PR[GP1:90,2] + 44.144;
   1:L PR[91] 10mm/sec CNT100;
   1:  PR[GP1:91,1] = PR[GP1:90,1] + 8.351;
   1:  PR[GP1:91,2] = PR[GP1:90,2] + 46.384;
   1:L PR[91] 10mm/sec CNT100;
   1:  PR[GP1:91,1] = PR[GP1:90,1] + 3.840;
   1:  PR[GP1:91,2] = PR[GP1:90,2] + 46.866;
   1:L PR[91] 10mm/sec CNT100;
   1:  PR[GP1:91,1] = PR[GP1:90,1] + -0.264;
   1:  PR[GP1:91,2] = PR[GP1:90,2] + 46.144;
   1:L PR[91] 10mm/sec CNT100;
   1:  PR[GP1:91,1] = PR[GP1:90,1] + -4.372;
   1:  PR[GP1:91,2] = PR[GP1:90,2] + 46.866;
   1:L PR[91] 10mm/sec CNT100;
   1:  PR[GP1:91,1] = PR[GP1:90,1] + -8.882;
   1:  PR[GP1:91,2] = PR[GP1:90,2] + 46.385;
   1:L PR[91] 10mm/sec CNT100;
   1:  PR[GP1:91,1] = PR[GP1:90,1] + -20.866;
   1:  PR[GP1:91,2] = PR[GP1:90,2] + 44.143;
   1:L PR[91] 10mm/sec CNT100;
   1:  PR[GP1:91,1] = PR[GP1:90,1] + -25.124;
   1:  PR[GP1:91,2] = PR[GP1:90,2] + 42.210;
   1:L PR[91] 10mm/sec CNT100;
   1:  PR[GP1:91,1] = PR[GP1:90,1] + -35.274;
   1:  PR[GP1:91,2] = PR[GP1:90,2] + 35.924;
   1:L PR[91] 10mm/sec CNT100;
   1:  PR[GP1:91,1] = PR[GP1:90,1] + -38.787;
   1:  PR[GP1:91,2] = PR[GP1:90,2] + 32.674;
   1:L PR[91] 10mm/sec CNT100;
   1:  PR[GP1:91,1] = PR[GP1:90,1] + -44.398;
   1:  PR[GP1:91,2] = PR[GP1:90,2] + 25.915;
   1:L PR[91] 10mm/sec CNT100;
   1:  PR[GP1:91,1] = PR[GP1:90,1] + -46.737;
   1:  PR[GP1:91,2] = PR[GP1:90,2] + 21.614;
   1:L PR[91] 10mm/sec CNT100;
   1:  PR[GP1:91,1] = PR[GP1:90,1] + -50.239;
   1:  PR[GP1:91,2] = PR[GP1:90,2] + 13.682;
   1:L PR[91] 10mm/sec CNT100;
   1:  PR[GP1:91,1] = PR[GP1:90,1] + -51.050;
   1:  PR[GP1:91,2] = PR[GP1:90,2] + 8.870;
   1:L PR[91] 10mm/sec CNT100;
   1:  PR[GP1:91,1] = PR[GP1:90,1] + -51.052;
   1:  PR[GP1:91,2] = PR[GP1:90,2] + 8.755;
   1:L PR[91] 10mm/sec CNT100;
   1:  PR[GP1:91,1] = PR[GP1:90,1] + -52.233;
   1:  PR[GP1:91,2] = PR[GP1:90,2] + 0.287;
   1:L PR[91] 10mm/sec CNT100;
   1:  PR[GP1:91,1] = PR[GP1:90,1] + -51.440;
   1:  PR[GP1:91,2] = PR[GP1:90,2] + -4.510;
   1:L PR[91] 10mm/sec CNT100;
   1:  PR[GP1:91,1] = PR[GP1:90,1] + -50.239;
   1:  PR[GP1:91,2] = PR[GP1:90,2] + -13.122;
   1:L PR[91] 10mm/sec CNT100;
   1:  PR[GP1:91,1] = PR[GP1:90,1] + -46.740;
   1:  PR[GP1:91,2] = PR[GP1:90,2] + -21.046;
   1:L PR[91] 10mm/sec CNT100;
   1:  PR[GP1:91,1] = PR[GP1:90,1] + -44.411;
   1:  PR[GP1:91,2] = PR[GP1:90,2] + -25.341;
   1:L PR[91] 10mm/sec CNT100;
   1:  PR[GP1:91,1] = PR[GP1:90,1] + -38.800;
   1:  PR[GP1:91,2] = PR[GP1:90,2] + -32.099;
   1:L PR[91] 10mm/sec CNT100;
   1:  PR[GP1:91,1] = PR[GP1:90,1] + -35.299;
   1:  PR[GP1:91,2] = PR[GP1:90,2] + -35.349;
   1:L PR[91] 10mm/sec CNT100;
   1:  PR[GP1:91,1] = PR[GP1:90,1] + -25.151;
   1:  PR[GP1:91,2] = PR[GP1:90,2] + -41.635;
   1:L PR[91] 10mm/sec CNT100;
   1:  PR[GP1:91,1] = PR[GP1:90,1] + -20.904;
   1:  PR[GP1:91,2] = PR[GP1:90,2] + -43.575;
   1:L PR[91] 10mm/sec CNT100;
   1:  PR[GP1:91,1] = PR[GP1:90,1] + -8.922;
   1:  PR[GP1:91,2] = PR[GP1:90,2] + -45.816;
   1:L PR[91] 10mm/sec CNT100;
   1:  PR[GP1:91,1] = PR[GP1:90,1] + -4.416;
   1:  PR[GP1:91,2] = PR[GP1:90,2] + -46.311;
   1:L PR[91] 10mm/sec CNT100;
   1:  PR[GP1:91,1] = PR[GP1:90,1] + -0.264;
   1:  PR[GP1:91,2] = PR[GP1:90,2] + -45.614;
   1:L PR[91] 10mm/sec CNT100;
   1:  PR[GP1:91,1] = PR[GP1:90,1] + 3.695;
   1:  PR[GP1:91,2] = PR[GP1:90,2] + -46.439;
   1:  PR[GP1:91,3] = PR[GP1:90,3] + 115.595;
   1:L PR[91] 10mm/sec CNT100;
   1:  PR[GP1:91,1] = PR[GP1:90,1] + 7.989;
   1:  PR[GP1:91,2] = PR[GP1:90,2] + -45.967;
   1:L PR[91] 10mm/sec CNT100;
   1:  PR[GP1:91,1] = PR[GP1:90,1] + 20.249;
   1:  PR[GP1:91,2] = PR[GP1:90,2] + -43.676;
   1:L PR[91] 10mm/sec CNT100;
   1:  PR[GP1:91,1] = PR[GP1:90,1] + 24.297;
   1:  PR[GP1:91,2] = PR[GP1:90,2] + -41.828;
   1:L PR[91] 10mm/sec CNT100;
   1:  PR[GP1:91,1] = PR[GP1:90,1] + 34.695;
   1:  PR[GP1:91,2] = PR[GP1:90,2] + -35.388;
   1:L PR[91] 10mm/sec CNT100;
   1:  PR[GP1:91,1] = PR[GP1:90,1] + 38.032;
   1:  PR[GP1:91,2] = PR[GP1:90,2] + -32.286;
   1:L PR[91] 10mm/sec CNT100;
   1:  PR[GP1:91,1] = PR[GP1:90,1] + 43.787;
   1:  PR[GP1:91,2] = PR[GP1:90,2] + -25.354;
   1:L PR[91] 10mm/sec CNT100;
   1:  PR[GP1:91,1] = PR[GP1:90,1] + 46.008;
   1:  PR[GP1:91,2] = PR[GP1:90,2] + -21.267;
   1:L PR[91] 10mm/sec CNT100;
   1:  PR[GP1:91,1] = PR[GP1:90,1] + 49.603;
   1:  PR[GP1:91,2] = PR[GP1:90,2] + -13.124;
   1:L PR[91] 10mm/sec CNT100;
   1:  PR[GP1:91,1] = PR[GP1:90,1] + 50.373;
   1:  PR[GP1:91,2] = PR[GP1:90,2] + -8.542;
   1:L PR[91] 10mm/sec CNT100;
   1:  PR[GP1:91,1] = PR[GP1:90,1] + 50.374;
   1:  PR[GP1:91,2] = PR[GP1:90,2] + -8.433;
   1:L PR[91] 10mm/sec CNT100;
   1:  PR[GP1:91,1] = PR[GP1:90,1] + 51.588;
   1:  PR[GP1:91,2] = PR[GP1:90,2] + 0.271;
   1:L PR[91] 10mm/sec CNT100;
   1:  PR[GP1:91,1] = PR[GP1:90,1] + 50.829;
   1:  PR[GP1:91,2] = PR[GP1:90,2] + 4.859;
   1:L PR[91] 10mm/sec CNT100;
   1:  PR[GP1:91,1] = PR[GP1:90,1] + 49.596;
   1:  PR[GP1:91,2] = PR[GP1:90,2] + 13.699;
   1:L PR[91] 10mm/sec CNT100;
   1:  PR[GP1:91,1] = PR[GP1:90,1] + 46.005;
   1:  PR[GP1:91,2] = PR[GP1:90,2] + 21.834;
   1:L PR[91] 10mm/sec CNT100;
   1:  PR[GP1:91,1] = PR[GP1:90,1] + 43.775;
   1:  PR[GP1:91,2] = PR[GP1:90,2] + 25.928;
   1:L PR[91] 10mm/sec CNT100;
   1:  PR[GP1:91,1] = PR[GP1:90,1] + 38.020;
   1:  PR[GP1:91,2] = PR[GP1:90,2] + 32.860;
   1:L PR[91] 10mm/sec CNT100;
   1:  PR[GP1:91,1] = PR[GP1:90,1] + 34.672;
   1:  PR[GP1:91,2] = PR[GP1:90,2] + 35.962;
   1:L PR[91] 10mm/sec CNT100;
   1:  PR[GP1:91,1] = PR[GP1:90,1] + 24.272;
   1:  PR[GP1:91,2] = PR[GP1:90,2] + 42.403;
   1:L PR[91] 10mm/sec CNT100;
   1:  PR[GP1:91,1] = PR[GP1:90,1] + 20.213;
   1:  PR[GP1:91,2] = PR[GP1:90,2] + 44.244;
   1:L PR[91] 10mm/sec CNT100;
   1:  PR[GP1:91,1] = PR[GP1:90,1] + 7.952;
   1:  PR[GP1:91,2] = PR[GP1:90,2] + 46.535;
   1:L PR[91] 10mm/sec CNT100;
   1:  PR[GP1:91,1] = PR[GP1:90,1] + 3.653;
   1:  PR[GP1:91,2] = PR[GP1:90,2] + 46.995;
   1:L PR[91] 10mm/sec CNT100;
   1:  PR[GP1:91,1] = PR[GP1:90,1] + -0.264;
   1:  PR[GP1:91,2] = PR[GP1:90,2] + 46.306;
   1:L PR[91] 10mm/sec CNT100;
   1:  PR[GP1:91,1] = PR[GP1:90,1] + -4.185;
   1:  PR[GP1:91,2] = PR[GP1:90,2] + 46.994;
   1:L PR[91] 10mm/sec CNT100;
   1:  PR[GP1:91,1] = PR[GP1:90,1] + -8.484;
   1:  PR[GP1:91,2] = PR[GP1:90,2] + 46.536;
   1:L PR[91] 10mm/sec CNT100;
   1:  PR[GP1:91,1] = PR[GP1:90,1] + -20.742;
   1:  PR[GP1:91,2] = PR[GP1:90,2] + 44.243;
   1:L PR[91] 10mm/sec CNT100;
   1:  PR[GP1:91,1] = PR[GP1:90,1] + -24.800;
   1:  PR[GP1:91,2] = PR[GP1:90,2] + 42.401;
   1:L PR[91] 10mm/sec CNT100;
   1:  PR[GP1:91,1] = PR[GP1:90,1] + -35.197;
   1:  PR[GP1:91,2] = PR[GP1:90,2] + 35.961;
   1:L PR[91] 10mm/sec CNT100;
   1:  PR[GP1:91,1] = PR[GP1:90,1] + -38.545;
   1:  PR[GP1:91,2] = PR[GP1:90,2] + 32.863;
   1:L PR[91] 10mm/sec CNT100;
   1:  PR[GP1:91,1] = PR[GP1:90,1] + -44.301;
   1:  PR[GP1:91,2] = PR[GP1:90,2] + 25.931;
   1:L PR[91] 10mm/sec CNT100;
   1:  PR[GP1:91,1] = PR[GP1:90,1] + -46.531;
   1:  PR[GP1:91,2] = PR[GP1:90,2] + 21.830;
   1:L PR[91] 10mm/sec CNT100;
   1:  PR[GP1:91,1] = PR[GP1:90,1] + -50.126;
   1:  PR[GP1:91,2] = PR[GP1:90,2] + 13.686;
   1:L PR[91] 10mm/sec CNT100;
   1:  PR[GP1:91,1] = PR[GP1:90,1] + -50.899;
   1:  PR[GP1:91,2] = PR[GP1:90,2] + 9.100;
   1:L PR[91] 10mm/sec CNT100;
   1:  PR[GP1:91,1] = PR[GP1:90,1] + -50.901;
   1:  PR[GP1:91,2] = PR[GP1:90,2] + 8.991;
   1:L PR[91] 10mm/sec CNT100;
   1:  PR[GP1:91,1] = PR[GP1:90,1] + -52.115;
   1:  PR[GP1:91,2] = PR[GP1:90,2] + 0.287;
   1:L PR[91] 10mm/sec CNT100;
   1:  PR[GP1:91,1] = PR[GP1:90,1] + -51.359;
   1:  PR[GP1:91,2] = PR[GP1:90,2] + -4.286;
   1:L PR[91] 10mm/sec CNT100;
   1:  PR[GP1:91,1] = PR[GP1:90,1] + -50.126;
   1:  PR[GP1:91,2] = PR[GP1:90,2] + -13.127;
   1:L PR[91] 10mm/sec CNT100;
   1:  PR[GP1:91,1] = PR[GP1:90,1] + -46.534;
   1:  PR[GP1:91,2] = PR[GP1:90,2] + -21.263;
   1:L PR[91] 10mm/sec CNT100;
   1:  PR[GP1:91,1] = PR[GP1:90,1] + -44.313;
   1:  PR[GP1:91,2] = PR[GP1:90,2] + -25.357;
   1:L PR[91] 10mm/sec CNT100;
   1:  PR[GP1:91,1] = PR[GP1:90,1] + -38.558;
   1:  PR[GP1:91,2] = PR[GP1:90,2] + -32.289;
   1:L PR[91] 10mm/sec CNT100;
   1:  PR[GP1:91,1] = PR[GP1:90,1] + -35.221;
   1:  PR[GP1:91,2] = PR[GP1:90,2] + -35.388;
   1:L PR[91] 10mm/sec CNT100;
   1:  PR[GP1:91,1] = PR[GP1:90,1] + -24.825;
   1:  PR[GP1:91,2] = PR[GP1:90,2] + -41.826;
   1:L PR[91] 10mm/sec CNT100;
   1:  PR[GP1:91,1] = PR[GP1:90,1] + -20.778;
   1:  PR[GP1:91,2] = PR[GP1:90,2] + -43.675;
   1:L PR[91] 10mm/sec CNT100;
   1:  PR[GP1:91,1] = PR[GP1:90,1] + -8.522;
   1:  PR[GP1:91,2] = PR[GP1:90,2] + -45.968;
   1:L PR[91] 10mm/sec CNT100;
   1:  PR[GP1:91,1] = PR[GP1:90,1] + -4.227;
   1:  PR[GP1:91,2] = PR[GP1:90,2] + -46.439;
   1:L PR[91] 10mm/sec CNT100;
   1:  PR[GP1:91,1] = PR[GP1:90,1] + -0.264;
   1:  PR[GP1:91,2] = PR[GP1:90,2] + -45.774;
   1:L PR[91] 10mm/sec CNT100;
   1:  PR[GP1:91,1] = PR[GP1:90,1] + 3.506;
   1:  PR[GP1:91,2] = PR[GP1:90,2] + -46.568;
   1:  PR[GP1:91,3] = PR[GP1:90,3] + 116.205;
   1:L PR[91] 10mm/sec CNT100;
   1:  PR[GP1:91,1] = PR[GP1:90,1] + 7.589;
   1:  PR[GP1:91,2] = PR[GP1:90,2] + -46.119;
   1:L PR[91] 10mm/sec CNT100;
   1:  PR[GP1:91,1] = PR[GP1:90,1] + 20.123;
   1:  PR[GP1:91,2] = PR[GP1:90,2] + -43.776;
   1:L PR[91] 10mm/sec CNT100;
   1:  PR[GP1:91,1] = PR[GP1:90,1] + 23.971;
   1:  PR[GP1:91,2] = PR[GP1:90,2] + -42.019;
   1:L PR[91] 10mm/sec CNT100;
   1:  PR[GP1:91,1] = PR[GP1:90,1] + 34.617;
   1:  PR[GP1:91,2] = PR[GP1:90,2] + -35.426;
   1:L PR[91] 10mm/sec CNT100;
   1:  PR[GP1:91,1] = PR[GP1:90,1] + 37.791;
   1:  PR[GP1:91,2] = PR[GP1:90,2] + -32.476;
   1:L PR[91] 10mm/sec CNT100;
   1:  PR[GP1:91,1] = PR[GP1:90,1] + 43.689;
   1:  PR[GP1:91,2] = PR[GP1:90,2] + -25.370;
   1:L PR[91] 10mm/sec CNT100;
   1:  PR[GP1:91,1] = PR[GP1:90,1] + 45.802;
   1:  PR[GP1:91,2] = PR[GP1:90,2] + -21.483;
   1:L PR[91] 10mm/sec CNT100;
   1:  PR[GP1:91,1] = PR[GP1:90,1] + 49.490;
   1:  PR[GP1:91,2] = PR[GP1:90,2] + -13.129;
   1:L PR[91] 10mm/sec CNT100;
   1:  PR[GP1:91,1] = PR[GP1:90,1] + 50.222;
   1:  PR[GP1:91,2] = PR[GP1:90,2] + -8.773;
   1:L PR[91] 10mm/sec CNT100;
   1:  PR[GP1:91,1] = PR[GP1:90,1] + 50.223;
   1:  PR[GP1:91,2] = PR[GP1:90,2] + -8.669;
   1:L PR[91] 10mm/sec CNT100;
   1:  PR[GP1:91,1] = PR[GP1:90,1] + 51.470;
   1:  PR[GP1:91,2] = PR[GP1:90,2] + 0.271;
   1:L PR[91] 10mm/sec CNT100;
   1:  PR[GP1:91,1] = PR[GP1:90,1] + 50.748;
   1:  PR[GP1:91,2] = PR[GP1:90,2] + 4.635;
   1:L PR[91] 10mm/sec CNT100;
   1:  PR[GP1:91,1] = PR[GP1:90,1] + 49.484;
   1:  PR[GP1:91,2] = PR[GP1:90,2] + 13.704;
   1:L PR[91] 10mm/sec CNT100;
   1:  PR[GP1:91,1] = PR[GP1:90,1] + 45.799;
   1:  PR[GP1:91,2] = PR[GP1:90,2] + 22.050;
   1:L PR[91] 10mm/sec CNT100;
   1:  PR[GP1:91,1] = PR[GP1:90,1] + 43.678;
   1:  PR[GP1:91,2] = PR[GP1:90,2] + 25.943;
   1:L PR[91] 10mm/sec CNT100;
   1:  PR[GP1:91,1] = PR[GP1:90,1] + 37.779;
   1:  PR[GP1:91,2] = PR[GP1:90,2] + 33.049;
   1:L PR[91] 10mm/sec CNT100;
   1:  PR[GP1:91,1] = PR[GP1:90,1] + 34.594;
   1:  PR[GP1:91,2] = PR[GP1:90,2] + 35.999;
   1:L PR[91] 10mm/sec CNT100;
   1:  PR[GP1:91,1] = PR[GP1:90,1] + 23.948;
   1:  PR[GP1:91,2] = PR[GP1:90,2] + 42.593;
   1:L PR[91] 10mm/sec CNT100;
   1:  PR[GP1:91,1] = PR[GP1:90,1] + 20.089;
   1:  PR[GP1:91,2] = PR[GP1:90,2] + 44.344;
   1:L PR[91] 10mm/sec CNT100;
   1:  PR[GP1:91,1] = PR[GP1:90,1] + 7.553;
   1:  PR[GP1:91,2] = PR[GP1:90,2] + 46.687;
   1:L PR[91] 10mm/sec CNT100;
   1:  PR[GP1:91,1] = PR[GP1:90,1] + 3.466;
   1:  PR[GP1:91,2] = PR[GP1:90,2] + 47.123;
   1:L PR[91] 10mm/sec CNT100;
   1:  PR[GP1:91,1] = PR[GP1:90,1] + -0.264;
   1:  PR[GP1:91,2] = PR[GP1:90,2] + 46.467;
   1:L PR[91] 10mm/sec CNT100;
   1:  PR[GP1:91,1] = PR[GP1:90,1] + -3.998;
   1:  PR[GP1:91,2] = PR[GP1:90,2] + 47.123;
   1:L PR[91] 10mm/sec CNT100;
   1:  PR[GP1:91,1] = PR[GP1:90,1] + -8.085;
   1:  PR[GP1:91,2] = PR[GP1:90,2] + 46.687;
   1:L PR[91] 10mm/sec CNT100;
   1:  PR[GP1:91,1] = PR[GP1:90,1] + -20.617;
   1:  PR[GP1:91,2] = PR[GP1:90,2] + 44.343;
   1:L PR[91] 10mm/sec CNT100;
   1:  PR[GP1:91,1] = PR[GP1:90,1] + -24.476;
   1:  PR[GP1:91,2] = PR[GP1:90,2] + 42.591;
   1:L PR[91] 10mm/sec CNT100;
   1:  PR[GP1:91,1] = PR[GP1:90,1] + -35.120;
   1:  PR[GP1:91,2] = PR[GP1:90,2] + 35.999;
   1:L PR[91] 10mm/sec CNT100;
   1:  PR[GP1:91,1] = PR[GP1:90,1] + -38.304;
   1:  PR[GP1:91,2] = PR[GP1:90,2] + 33.053;
   1:L PR[91] 10mm/sec CNT100;
   1:  PR[GP1:91,1] = PR[GP1:90,1] + -44.204;
   1:  PR[GP1:91,2] = PR[GP1:90,2] + 25.947;
   1:L PR[91] 10mm/sec CNT100;
   1:  PR[GP1:91,1] = PR[GP1:90,1] + -46.325;
   1:  PR[GP1:91,2] = PR[GP1:90,2] + 22.046;
   1:L PR[91] 10mm/sec CNT100;
   1:  PR[GP1:91,1] = PR[GP1:90,1] + -50.013;
   1:  PR[GP1:91,2] = PR[GP1:90,2] + 13.691;
   1:L PR[91] 10mm/sec CNT100;
   1:  PR[GP1:91,1] = PR[GP1:90,1] + -50.749;
   1:  PR[GP1:91,2] = PR[GP1:90,2] + 9.331;
   1:L PR[91] 10mm/sec CNT100;
   1:  PR[GP1:91,1] = PR[GP1:90,1] + -50.750;
   1:  PR[GP1:91,2] = PR[GP1:90,2] + 9.228;
   1:L PR[91] 10mm/sec CNT100;
   1:  PR[GP1:91,1] = PR[GP1:90,1] + -51.997;
   1:  PR[GP1:91,2] = PR[GP1:90,2] + 0.287;
   1:L PR[91] 10mm/sec CNT100;
   1:  PR[GP1:91,1] = PR[GP1:90,1] + -51.278;
   1:  PR[GP1:91,2] = PR[GP1:90,2] + -4.063;
   1:L PR[91] 10mm/sec CNT100;
   1:  PR[GP1:91,1] = PR[GP1:90,1] + -50.013;
   1:  PR[GP1:91,2] = PR[GP1:90,2] + -13.132;
   1:L PR[91] 10mm/sec CNT100;
   1:  PR[GP1:91,1] = PR[GP1:90,1] + -46.328;
   1:  PR[GP1:91,2] = PR[GP1:90,2] + -21.479;
   1:L PR[91] 10mm/sec CNT100;
   1:  PR[GP1:91,1] = PR[GP1:90,1] + -44.215;
   1:  PR[GP1:91,2] = PR[GP1:90,2] + -25.374;
   1:L PR[91] 10mm/sec CNT100;
   1:  PR[GP1:91,1] = PR[GP1:90,1] + -38.316;
   1:  PR[GP1:91,2] = PR[GP1:90,2] + -32.480;
   1:L PR[91] 10mm/sec CNT100;
   1:  PR[GP1:91,1] = PR[GP1:90,1] + -35.143;
   1:  PR[GP1:91,2] = PR[GP1:90,2] + -35.426;
   1:L PR[91] 10mm/sec CNT100;
   1:  PR[GP1:91,1] = PR[GP1:90,1] + -24.500;
   1:  PR[GP1:91,2] = PR[GP1:90,2] + -42.018;
   1:L PR[91] 10mm/sec CNT100;
   1:  PR[GP1:91,1] = PR[GP1:90,1] + -20.651;
   1:  PR[GP1:91,2] = PR[GP1:90,2] + -43.776;
   1:L PR[91] 10mm/sec CNT100;
   1:  PR[GP1:91,1] = PR[GP1:90,1] + -8.121;
   1:  PR[GP1:91,2] = PR[GP1:90,2] + -46.119;
   1:L PR[91] 10mm/sec CNT100;
   1:  PR[GP1:91,1] = PR[GP1:90,1] + -4.038;
   1:  PR[GP1:91,2] = PR[GP1:90,2] + -46.567;
   1:L PR[91] 10mm/sec CNT100;
   1:  PR[GP1:91,1] = PR[GP1:90,1] + -0.264;
   1:  PR[GP1:91,2] = PR[GP1:90,2] + -45.935;
   1:L PR[91] 10mm/sec CNT100;
   1:  PR[GP1:91,1] = PR[GP1:90,1] + 3.316;
   1:  PR[GP1:91,2] = PR[GP1:90,2] + -46.696;
   1:  PR[GP1:91,3] = PR[GP1:90,3] + 116.815;
   1:L PR[91] 10mm/sec CNT100;
   1:  PR[GP1:91,1] = PR[GP1:90,1] + 7.188;
   1:  PR[GP1:91,2] = PR[GP1:90,2] + -46.271;
   1:L PR[91] 10mm/sec CNT100;
   1:  PR[GP1:91,1] = PR[GP1:90,1] + 19.997;
   1:  PR[GP1:91,2] = PR[GP1:90,2] + -43.877;
   1:L PR[91] 10mm/sec CNT100;
   1:  PR[GP1:91,1] = PR[GP1:90,1] + 23.646;
   1:  PR[GP1:91,2] = PR[GP1:90,2] + -42.211;
   1:L PR[91] 10mm/sec CNT100;
   1:  PR[GP1:91,1] = PR[GP1:90,1] + 34.539;
   1:  PR[GP1:91,2] = PR[GP1:90,2] + -35.464;
   1:L PR[91] 10mm/sec CNT100;
   1:  PR[GP1:91,1] = PR[GP1:90,1] + 37.549;
   1:  PR[GP1:91,2] = PR[GP1:90,2] + -32.667;
   1:L PR[91] 10mm/sec CNT100;
   1:  PR[GP1:91,1] = PR[GP1:90,1] + 43.592;
   1:  PR[GP1:91,2] = PR[GP1:90,2] + -25.387;
   1:L PR[91] 10mm/sec CNT100;
   1:  PR[GP1:91,1] = PR[GP1:90,1] + 45.596;
   1:  PR[GP1:91,2] = PR[GP1:90,2] + -21.699;
   1:L PR[91] 10mm/sec CNT100;
   1:  PR[GP1:91,1] = PR[GP1:90,1] + 49.377;
   1:  PR[GP1:91,2] = PR[GP1:90,2] + -13.134;
   1:L PR[91] 10mm/sec CNT100;
   1:  PR[GP1:91,1] = PR[GP1:90,1] + 50.071;
   1:  PR[GP1:91,2] = PR[GP1:90,2] + -9.003;
   1:L PR[91] 10mm/sec CNT100;
   1:  PR[GP1:91,1] = PR[GP1:90,1] + 50.072;
   1:  PR[GP1:91,2] = PR[GP1:90,2] + -8.905;
   1:L PR[91] 10mm/sec CNT100;
   1:  PR[GP1:91,1] = PR[GP1:90,1] + 51.352;
   1:  PR[GP1:91,2] = PR[GP1:90,2] + 0.271;
   1:L PR[91] 10mm/sec CNT100;
   1:  PR[GP1:91,1] = PR[GP1:90,1] + 50.668;
   1:  PR[GP1:91,2] = PR[GP1:90,2] + 4.410;
   1:L PR[91] 10mm/sec CNT100;
   1:  PR[GP1:91,1] = PR[GP1:90,1] + 49.371;
   1:  PR[GP1:91,2] = PR[GP1:90,2] + 13.708;
   1:L PR[91] 10mm/sec CNT100;
   1:  PR[GP1:91,1] = PR[GP1:90,1] + 45.593;
   1:  PR[GP1:91,2] = PR[GP1:90,2] + 22.266;
   1:L PR[91] 10mm/sec CNT100;
   1:  PR[GP1:91,1] = PR[GP1:90,1] + 43.581;
   1:  PR[GP1:91,2] = PR[GP1:90,2] + 25.959;
   1:L PR[91] 10mm/sec CNT100;
   1:  PR[GP1:91,1] = PR[GP1:90,1] + 37.537;
   1:  PR[GP1:91,2] = PR[GP1:90,2] + 33.239;
   1:L PR[91] 10mm/sec CNT100;
   1:  PR[GP1:91,1] = PR[GP1:90,1] + 34.517;
   1:  PR[GP1:91,2] = PR[GP1:90,2] + 36.037;
   1:L PR[91] 10mm/sec CNT100;
   1:  PR[GP1:91,1] = PR[GP1:90,1] + 23.624;
   1:  PR[GP1:91,2] = PR[GP1:90,2] + 42.784;
   1:L PR[91] 10mm/sec CNT100;
   1:  PR[GP1:91,1] = PR[GP1:90,1] + 19.964;
   1:  PR[GP1:91,2] = PR[GP1:90,2] + 44.443;
   1:L PR[91] 10mm/sec CNT100;
   1:  PR[GP1:91,1] = PR[GP1:90,1] + 7.155;
   1:  PR[GP1:91,2] = PR[GP1:90,2] + 46.838;
   1:L PR[91] 10mm/sec CNT100;
   1:  PR[GP1:91,1] = PR[GP1:90,1] + 3.278;
   1:  PR[GP1:91,2] = PR[GP1:90,2] + 47.252;
   1:L PR[91] 10mm/sec CNT100;
   1:  PR[GP1:91,1] = PR[GP1:90,1] + -0.264;
   1:  PR[GP1:91,2] = PR[GP1:90,2] + 46.629;
   1:L PR[91] 10mm/sec CNT100;
   1:  PR[GP1:91,1] = PR[GP1:90,1] + -3.811;
   1:  PR[GP1:91,2] = PR[GP1:90,2] + 47.252;
   1:L PR[91] 10mm/sec CNT100;
   1:  PR[GP1:91,1] = PR[GP1:90,1] + -7.687;
   1:  PR[GP1:91,2] = PR[GP1:90,2] + 46.838;
   1:L PR[91] 10mm/sec CNT100;
   1:  PR[GP1:91,1] = PR[GP1:90,1] + -20.493;
   1:  PR[GP1:91,2] = PR[GP1:90,2] + 44.443;
   1:L PR[91] 10mm/sec CNT100;
   1:  PR[GP1:91,1] = PR[GP1:90,1] + -24.152;
   1:  PR[GP1:91,2] = PR[GP1:90,2] + 42.782;
   1:L PR[91] 10mm/sec CNT100;
   1:  PR[GP1:91,1] = PR[GP1:90,1] + -35.043;
   1:  PR[GP1:91,2] = PR[GP1:90,2] + 36.037;
   1:L PR[91] 10mm/sec CNT100;
   1:  PR[GP1:91,1] = PR[GP1:90,1] + -38.063;
   1:  PR[GP1:91,2] = PR[GP1:90,2] + 33.242;
   1:L PR[91] 10mm/sec CNT100;
   1:  PR[GP1:91,1] = PR[GP1:90,1] + -44.106;
   1:  PR[GP1:91,2] = PR[GP1:90,2] + 25.962;
   1:L PR[91] 10mm/sec CNT100;
   1:  PR[GP1:91,1] = PR[GP1:90,1] + -46.119;
   1:  PR[GP1:91,2] = PR[GP1:90,2] + 22.262;
   1:L PR[91] 10mm/sec CNT100;
   1:  PR[GP1:91,1] = PR[GP1:90,1] + -49.900;
   1:  PR[GP1:91,2] = PR[GP1:90,2] + 13.696;
   1:L PR[91] 10mm/sec CNT100;
   1:  PR[GP1:91,1] = PR[GP1:90,1] + -50.598;
   1:  PR[GP1:91,2] = PR[GP1:90,2] + 9.562;
   1:L PR[91] 10mm/sec CNT100;
   1:  PR[GP1:91,1] = PR[GP1:90,1] + -50.599;
   1:  PR[GP1:91,2] = PR[GP1:90,2] + 9.464;
   1:L PR[91] 10mm/sec CNT100;
   1:  PR[GP1:91,1] = PR[GP1:90,1] + -51.879;
   1:  PR[GP1:91,2] = PR[GP1:90,2] + 0.287;
   1:L PR[91] 10mm/sec CNT100;
   1:  PR[GP1:91,1] = PR[GP1:90,1] + -51.197;
   1:  PR[GP1:91,2] = PR[GP1:90,2] + -3.840;
   1:L PR[91] 10mm/sec CNT100;
   1:  PR[GP1:91,1] = PR[GP1:90,1] + -49.900;
   1:  PR[GP1:91,2] = PR[GP1:90,2] + -13.137;
   1:L PR[91] 10mm/sec CNT100;
   1:  PR[GP1:91,1] = PR[GP1:90,1] + -46.122;
   1:  PR[GP1:91,2] = PR[GP1:90,2] + -21.696;
   1:L PR[91] 10mm/sec CNT100;
   1:  PR[GP1:91,1] = PR[GP1:90,1] + -44.117;
   1:  PR[GP1:91,2] = PR[GP1:90,2] + -25.390;
   1:L PR[91] 10mm/sec CNT100;
   1:  PR[GP1:91,1] = PR[GP1:90,1] + -38.074;
   1:  PR[GP1:91,2] = PR[GP1:90,2] + -32.670;
   1:L PR[91] 10mm/sec CNT100;
   1:  PR[GP1:91,1] = PR[GP1:90,1] + -35.064;
   1:  PR[GP1:91,2] = PR[GP1:90,2] + -35.464;
   1:L PR[91] 10mm/sec CNT100;
   1:  PR[GP1:91,1] = PR[GP1:90,1] + -24.175;
   1:  PR[GP1:91,2] = PR[GP1:90,2] + -42.209;
   1:L PR[91] 10mm/sec CNT100;
   1:  PR[GP1:91,1] = PR[GP1:90,1] + -20.525;
   1:  PR[GP1:91,2] = PR[GP1:90,2] + -43.876;
   1:L PR[91] 10mm/sec CNT100;
   1:  PR[GP1:91,1] = PR[GP1:90,1] + -7.721;
   1:  PR[GP1:91,2] = PR[GP1:90,2] + -46.271;
   1:L PR[91] 10mm/sec CNT100;
   1:  PR[GP1:91,1] = PR[GP1:90,1] + -3.849;
   1:  PR[GP1:91,2] = PR[GP1:90,2] + -46.696;
   1:L PR[91] 10mm/sec CNT100;
   1:  PR[GP1:91,1] = PR[GP1:90,1] + -0.264;
   1:  PR[GP1:91,2] = PR[GP1:90,2] + -46.095;
   1:L PR[91] 10mm/sec CNT100;
   1:  PR[GP1:91,1] = PR[GP1:90,1] + 3.127;
   1:  PR[GP1:91,2] = PR[GP1:90,2] + -46.824;
   1:  PR[GP1:91,3] = PR[GP1:90,3] + 117.425;
   1:L PR[91] 10mm/sec CNT100;
   1:  PR[GP1:91,1] = PR[GP1:90,1] + 6.788;
   1:  PR[GP1:91,2] = PR[GP1:90,2] + -46.422;
   1:L PR[91] 10mm/sec CNT100;
   1:  PR[GP1:91,1] = PR[GP1:90,1] + 19.870;
   1:  PR[GP1:91,2] = PR[GP1:90,2] + -43.977;
   1:L PR[91] 10mm/sec CNT100;
   1:  PR[GP1:91,1] = PR[GP1:90,1] + 23.321;
   1:  PR[GP1:91,2] = PR[GP1:90,2] + -42.402;
   1:L PR[91] 10mm/sec CNT100;
   1:  PR[GP1:91,1] = PR[GP1:90,1] + 34.460;
   1:  PR[GP1:91,2] = PR[GP1:90,2] + -35.503;
   1:L PR[91] 10mm/sec CNT100;
   1:  PR[GP1:91,1] = PR[GP1:90,1] + 37.307;
   1:  PR[GP1:91,2] = PR[GP1:90,2] + -32.857;
   1:L PR[91] 10mm/sec CNT100;
   1:  PR[GP1:91,1] = PR[GP1:90,1] + 43.494;
   1:  PR[GP1:91,2] = PR[GP1:90,2] + -25.404;
   1:L PR[91] 10mm/sec CNT100;
   1:  PR[GP1:91,1] = PR[GP1:90,1] + 45.390;
   1:  PR[GP1:91,2] = PR[GP1:90,2] + -21.916;
   1:L PR[91] 10mm/sec CNT100;
   1:  PR[GP1:91,1] = PR[GP1:90,1] + 49.264;
   1:  PR[GP1:91,2] = PR[GP1:90,2] + -13.139;
   1:L PR[91] 10mm/sec CNT100;
   1:  PR[GP1:91,1] = PR[GP1:90,1] + 49.920;
   1:  PR[GP1:91,2] = PR[GP1:90,2] + -9.234;
   1:L PR[91] 10mm/sec CNT100;
   1:  PR[GP1:91,1] = PR[GP1:90,1] + 49.922;
   1:  PR[GP1:91,2] = PR[GP1:90,2] + -9.142;
   1:L PR[91] 10mm/sec CNT100;
   1:  PR[GP1:91,1] = PR[GP1:90,1] + 51.234;
   1:  PR[GP1:91,2] = PR[GP1:90,2] + 0.271;
   1:L PR[91] 10mm/sec CNT100;
   1:  PR[GP1:91,1] = PR[GP1:90,1] + 50.587;
   1:  PR[GP1:91,2] = PR[GP1:90,2] + 4.186;
   1:L PR[91] 10mm/sec CNT100;
   1:  PR[GP1:91,1] = PR[GP1:90,1] + 49.258;
   1:  PR[GP1:91,2] = PR[GP1:90,2] + 13.713;
   1:L PR[91] 10mm/sec CNT100;
   1:  PR[GP1:91,1] = PR[GP1:90,1] + 45.387;
   1:  PR[GP1:91,2] = PR[GP1:90,2] + 22.482;
   1:L PR[91] 10mm/sec CNT100;
   1:  PR[GP1:91,1] = PR[GP1:90,1] + 43.483;
   1:  PR[GP1:91,2] = PR[GP1:90,2] + 25.975;
   1:L PR[91] 10mm/sec CNT100;
   1:  PR[GP1:91,1] = PR[GP1:90,1] + 37.296;
   1:  PR[GP1:91,2] = PR[GP1:90,2] + 33.429;
   1:L PR[91] 10mm/sec CNT100;
   1:  PR[GP1:91,1] = PR[GP1:90,1] + 34.440;
   1:  PR[GP1:91,2] = PR[GP1:90,2] + 36.074;
   1:L PR[91] 10mm/sec CNT100;
   1:  PR[GP1:91,1] = PR[GP1:90,1] + 23.299;
   1:  PR[GP1:91,2] = PR[GP1:90,2] + 42.974;
   1:L PR[91] 10mm/sec CNT100;
   1:  PR[GP1:91,1] = PR[GP1:90,1] + 19.840;
   1:  PR[GP1:91,2] = PR[GP1:90,2] + 44.543;
   1:L PR[91] 10mm/sec CNT100;
   1:  PR[GP1:91,1] = PR[GP1:90,1] + 6.756;
   1:  PR[GP1:91,2] = PR[GP1:90,2] + 46.989;
   1:L PR[91] 10mm/sec CNT100;
   1:  PR[GP1:91,1] = PR[GP1:90,1] + 3.091;
   1:  PR[GP1:91,2] = PR[GP1:90,2] + 47.380;
   1:L PR[91] 10mm/sec CNT100;
   1:  PR[GP1:91,1] = PR[GP1:90,1] + -0.264;
   1:  PR[GP1:91,2] = PR[GP1:90,2] + 46.790;
   1:L PR[91] 10mm/sec CNT100;
   1:  PR[GP1:91,1] = PR[GP1:90,1] + -3.624;
   1:  PR[GP1:91,2] = PR[GP1:90,2] + 47.380;
   1:L PR[91] 10mm/sec CNT100;
   1:  PR[GP1:91,1] = PR[GP1:90,1] + -7.288;
   1:  PR[GP1:91,2] = PR[GP1:90,2] + 46.989;
   1:L PR[91] 10mm/sec CNT100;
   1:  PR[GP1:91,1] = PR[GP1:90,1] + -20.368;
   1:  PR[GP1:91,2] = PR[GP1:90,2] + 44.543;
   1:L PR[91] 10mm/sec CNT100;
   1:  PR[GP1:91,1] = PR[GP1:90,1] + -23.828;
   1:  PR[GP1:91,2] = PR[GP1:90,2] + 42.972;
   1:L PR[91] 10mm/sec CNT100;
   1:  PR[GP1:91,1] = PR[GP1:90,1] + -34.965;
   1:  PR[GP1:91,2] = PR[GP1:90,2] + 36.074;
   1:L PR[91] 10mm/sec CNT100;
   1:  PR[GP1:91,1] = PR[GP1:90,1] + -37.821;
   1:  PR[GP1:91,2] = PR[GP1:90,2] + 33.432;
   1:L PR[91] 10mm/sec CNT100;
   1:  PR[GP1:91,1] = PR[GP1:90,1] + -44.009;
   1:  PR[GP1:91,2] = PR[GP1:90,2] + 25.978;
   1:L PR[91] 10mm/sec CNT100;
   1:  PR[GP1:91,1] = PR[GP1:90,1] + -45.913;
   1:  PR[GP1:91,2] = PR[GP1:90,2] + 22.478;
   1:L PR[91] 10mm/sec CNT100;
   1:  PR[GP1:91,1] = PR[GP1:90,1] + -49.788;
   1:  PR[GP1:91,2] = PR[GP1:90,2] + 13.701;
   1:L PR[91] 10mm/sec CNT100;
   1:  PR[GP1:91,1] = PR[GP1:90,1] + -50.447;
   1:  PR[GP1:91,2] = PR[GP1:90,2] + 9.792;
   1:L PR[91] 10mm/sec CNT100;
   1:  PR[GP1:91,1] = PR[GP1:90,1] + -50.448;
   1:  PR[GP1:91,2] = PR[GP1:90,2] + 9.700;
   1:L PR[91] 10mm/sec CNT100;
   1:  PR[GP1:91,1] = PR[GP1:90,1] + -51.761;
   1:  PR[GP1:91,2] = PR[GP1:90,2] + 0.287;
   1:L PR[91] 10mm/sec CNT100;
   1:  PR[GP1:91,1] = PR[GP1:90,1] + -51.116;
   1:  PR[GP1:91,2] = PR[GP1:90,2] + -3.616;
   1:L PR[91] 10mm/sec CNT100;
   1:  PR[GP1:91,1] = PR[GP1:90,1] + -49.787;
   1:  PR[GP1:91,2] = PR[GP1:90,2] + -13.143;
   1:L PR[91] 10mm/sec CNT100;
   1:  PR[GP1:91,1] = PR[GP1:90,1] + -45.916;
   1:  PR[GP1:91,2] = PR[GP1:90,2] + -21.912;
   1:L PR[91] 10mm/sec CNT100;
   1:  PR[GP1:91,1] = PR[GP1:90,1] + -44.020;
   1:  PR[GP1:91,2] = PR[GP1:90,2] + -25.407;
   1:L PR[91] 10mm/sec CNT100;
   1:  PR[GP1:91,1] = PR[GP1:90,1] + -37.832;
   1:  PR[GP1:91,2] = PR[GP1:90,2] + -32.860;
   1:L PR[91] 10mm/sec CNT100;
   1:  PR[GP1:91,1] = PR[GP1:90,1] + -34.986;
   1:  PR[GP1:91,2] = PR[GP1:90,2] + -35.503;
   1:L PR[91] 10mm/sec CNT100;
   1:  PR[GP1:91,1] = PR[GP1:90,1] + -23.849;
   1:  PR[GP1:91,2] = PR[GP1:90,2] + -42.400;
   1:L PR[91] 10mm/sec CNT100;
   1:  PR[GP1:91,1] = PR[GP1:90,1] + -20.399;
   1:  PR[GP1:91,2] = PR[GP1:90,2] + -43.976;
   1:L PR[91] 10mm/sec CNT100;
   1:  PR[GP1:91,1] = PR[GP1:90,1] + -7.320;
   1:  PR[GP1:91,2] = PR[GP1:90,2] + -46.423;
   1:L PR[91] 10mm/sec CNT100;
   1:  PR[GP1:91,1] = PR[GP1:90,1] + -3.659;
   1:  PR[GP1:91,2] = PR[GP1:90,2] + -46.824;
   1:L PR[91] 10mm/sec CNT100;
   1:  PR[GP1:91,1] = PR[GP1:90,1] + -0.264;
   1:  PR[GP1:91,2] = PR[GP1:90,2] + -46.255;
   1:L PR[91] 10mm/sec CNT100;
   1:  PR[GP1:91,1] = PR[GP1:90,1] + 2.938;
   1:  PR[GP1:91,2] = PR[GP1:90,2] + -46.953;
   1:  PR[GP1:91,3] = PR[GP1:90,3] + 118.035;
   1:L PR[91] 10mm/sec CNT100;
   1:  PR[GP1:91,1] = PR[GP1:90,1] + 6.387;
   1:  PR[GP1:91,2] = PR[GP1:90,2] + -46.574;
   1:L PR[91] 10mm/sec CNT100;
   1:  PR[GP1:91,1] = PR[GP1:90,1] + 19.744;
   1:  PR[GP1:91,2] = PR[GP1:90,2] + -44.077;
   1:L PR[91] 10mm/sec CNT100;
   1:  PR[GP1:91,1] = PR[GP1:90,1] + 22.995;
   1:  PR[GP1:91,2] = PR[GP1:90,2] + -42.593;
   1:L PR[91] 10mm/sec CNT100;
   1:  PR[GP1:91,1] = PR[GP1:90,1] + 34.382;
   1:  PR[GP1:91,2] = PR[GP1:90,2] + -35.541;
   1:L PR[91] 10mm/sec CNT100;
   1:  PR[GP1:91,1] = PR[GP1:90,1] + 37.065;
   1:  PR[GP1:91,2] = PR[GP1:90,2] + -33.047;
   1:L PR[91] 10mm/sec CNT100;
   1:  PR[GP1:91,1] = PR[GP1:90,1] + 43.396;
   1:  PR[GP1:91,2] = PR[GP1:90,2] + -25.420;
   1:L PR[91] 10mm/sec CNT100;
   1:  PR[GP1:91,1] = PR[GP1:90,1] + 45.183;
   1:  PR[GP1:91,2] = PR[GP1:90,2] + -22.132;
   1:L PR[91] 10mm/sec CNT100;
   1:  PR[GP1:91,1] = PR[GP1:90,1] + 49.151;
   1:  PR[GP1:91,2] = PR[GP1:90,2] + -13.144;
   1:L PR[91] 10mm/sec CNT100;
   1:  PR[GP1:91,1] = PR[GP1:90,1] + 49.770;
   1:  PR[GP1:91,2] = PR[GP1:90,2] + -9.465;
   1:L PR[91] 10mm/sec CNT100;
   1:  PR[GP1:91,1] = PR[GP1:90,1] + 49.771;
   1:  PR[GP1:91,2] = PR[GP1:90,2] + -9.378;
   1:L PR[91] 10mm/sec CNT100;
   1:  PR[GP1:91,1] = PR[GP1:90,1] + 51.116;
   1:  PR[GP1:91,2] = PR[GP1:90,2] + 0.271;
   1:L PR[91] 10mm/sec CNT100;
   1:  PR[GP1:91,1] = PR[GP1:90,1] + 50.506;
   1:  PR[GP1:91,2] = PR[GP1:90,2] + 3.962;
   1:L PR[91] 10mm/sec CNT100;
   1:  PR[GP1:91,1] = PR[GP1:90,1] + 49.145;
   1:  PR[GP1:91,2] = PR[GP1:90,2] + 13.717;
   1:L PR[91] 10mm/sec CNT100;
   1:  PR[GP1:91,1] = PR[GP1:90,1] + 45.181;
   1:  PR[GP1:91,2] = PR[GP1:90,2] + 22.697;
   1:L PR[91] 10mm/sec CNT100;
   1:  PR[GP1:91,1] = PR[GP1:90,1] + 43.386;
   1:  PR[GP1:91,2] = PR[GP1:90,2] + 25.991;
   1:L PR[91] 10mm/sec CNT100;
   1:  PR[GP1:91,1] = PR[GP1:90,1] + 37.055;
   1:  PR[GP1:91,2] = PR[GP1:90,2] + 33.618;
   1:L PR[91] 10mm/sec CNT100;
   1:  PR[GP1:91,1] = PR[GP1:90,1] + 34.363;
   1:  PR[GP1:91,2] = PR[GP1:90,2] + 36.112;
   1:L PR[91] 10mm/sec CNT100;
   1:  PR[GP1:91,1] = PR[GP1:90,1] + 22.975;
   1:  PR[GP1:91,2] = PR[GP1:90,2] + 43.164;
   1:L PR[91] 10mm/sec CNT100;
   1:  PR[GP1:91,1] = PR[GP1:90,1] + 19.715;
   1:  PR[GP1:91,2] = PR[GP1:90,2] + 44.643;
   1:L PR[91] 10mm/sec CNT100;
   1:  PR[GP1:91,1] = PR[GP1:90,1] + 6.357;
   1:  PR[GP1:91,2] = PR[GP1:90,2] + 47.140;
   1:L PR[91] 10mm/sec CNT100;
   1:  PR[GP1:91,1] = PR[GP1:90,1] + 2.904;
   1:  PR[GP1:91,2] = PR[GP1:90,2] + 47.509;
   1:L PR[91] 10mm/sec CNT100;
   1:  PR[GP1:91,1] = PR[GP1:90,1] + -0.264;
   1:  PR[GP1:91,2] = PR[GP1:90,2] + 46.952;
   1:L PR[91] 10mm/sec CNT100;
   1:  PR[GP1:91,1] = PR[GP1:90,1] + -3.436;
   1:  PR[GP1:91,2] = PR[GP1:90,2] + 47.509;
   1:L PR[91] 10mm/sec CNT100;
   1:  PR[GP1:91,1] = PR[GP1:90,1] + -6.890;
   1:  PR[GP1:91,2] = PR[GP1:90,2] + 47.140;
   1:L PR[91] 10mm/sec CNT100;
   1:  PR[GP1:91,1] = PR[GP1:90,1] + -20.244;
   1:  PR[GP1:91,2] = PR[GP1:90,2] + 44.643;
   1:L PR[91] 10mm/sec CNT100;
   1:  PR[GP1:91,1] = PR[GP1:90,1] + -23.504;
   1:  PR[GP1:91,2] = PR[GP1:90,2] + 43.163;
   1:L PR[91] 10mm/sec CNT100;
   1:  PR[GP1:91,1] = PR[GP1:90,1] + -34.888;
   1:  PR[GP1:91,2] = PR[GP1:90,2] + 36.112;
   1:L PR[91] 10mm/sec CNT100;
   1:  PR[GP1:91,1] = PR[GP1:90,1] + -37.580;
   1:  PR[GP1:91,2] = PR[GP1:90,2] + 33.621;
   1:L PR[91] 10mm/sec CNT100;
   1:  PR[GP1:91,1] = PR[GP1:90,1] + -43.912;
   1:  PR[GP1:91,2] = PR[GP1:90,2] + 25.994;
   1:L PR[91] 10mm/sec CNT100;
   1:  PR[GP1:91,1] = PR[GP1:90,1] + -45.707;
   1:  PR[GP1:91,2] = PR[GP1:90,2] + 22.694;
   1:L PR[91] 10mm/sec CNT100;
   1:  PR[GP1:91,1] = PR[GP1:90,1] + -49.675;
   1:  PR[GP1:91,2] = PR[GP1:90,2] + 13.706;
   1:L PR[91] 10mm/sec CNT100;
   1:  PR[GP1:91,1] = PR[GP1:90,1] + -50.296;
   1:  PR[GP1:91,2] = PR[GP1:90,2] + 10.023;
   1:L PR[91] 10mm/sec CNT100;
   1:  PR[GP1:91,1] = PR[GP1:90,1] + -50.297;
   1:  PR[GP1:91,2] = PR[GP1:90,2] + 9.937;
   1:L PR[91] 10mm/sec CNT100;
   1:  PR[GP1:91,1] = PR[GP1:90,1] + -51.643;
   1:  PR[GP1:91,2] = PR[GP1:90,2] + 0.287;
   1:L PR[91] 10mm/sec CNT100;
   1:  PR[GP1:91,1] = PR[GP1:90,1] + -51.035;
   1:  PR[GP1:91,2] = PR[GP1:90,2] + -3.393;
   1:L PR[91] 10mm/sec CNT100;
   1:  PR[GP1:91,1] = PR[GP1:90,1] + -49.674;
   1:  PR[GP1:91,2] = PR[GP1:90,2] + -13.148;
   1:L PR[91] 10mm/sec CNT100;
   1:  PR[GP1:91,1] = PR[GP1:90,1] + -45.709;
   1:  PR[GP1:91,2] = PR[GP1:90,2] + -22.129;
   1:L PR[91] 10mm/sec CNT100;
   1:  PR[GP1:91,1] = PR[GP1:90,1] + -43.922;
   1:  PR[GP1:91,2] = PR[GP1:90,2] + -25.423;
   1:L PR[91] 10mm/sec CNT100;
   1:  PR[GP1:91,1] = PR[GP1:90,1] + -37.590;
   1:  PR[GP1:91,2] = PR[GP1:90,2] + -33.050;
   1:L PR[91] 10mm/sec CNT100;
   1:  PR[GP1:91,1] = PR[GP1:90,1] + -34.908;
   1:  PR[GP1:91,2] = PR[GP1:90,2] + -35.541;
   1:L PR[91] 10mm/sec CNT100;
   1:  PR[GP1:91,1] = PR[GP1:90,1] + -23.524;
   1:  PR[GP1:91,2] = PR[GP1:90,2] + -42.592;
   1:L PR[91] 10mm/sec CNT100;
   1:  PR[GP1:91,1] = PR[GP1:90,1] + -20.273;
   1:  PR[GP1:91,2] = PR[GP1:90,2] + -44.077;
   1:L PR[91] 10mm/sec CNT100;
   1:  PR[GP1:91,1] = PR[GP1:90,1] + -6.920;
   1:  PR[GP1:91,2] = PR[GP1:90,2] + -46.574;
   1:L PR[91] 10mm/sec CNT100;
   1:  PR[GP1:91,1] = PR[GP1:90,1] + -3.470;
   1:  PR[GP1:91,2] = PR[GP1:90,2] + -46.953;
   1:L PR[91] 10mm/sec CNT100;
   1:  PR[GP1:91,1] = PR[GP1:90,1] + -0.264;
   1:  PR[GP1:91,2] = PR[GP1:90,2] + -46.415;
   1:L PR[91] 10mm/sec CNT100;
   1:  PR[GP1:91,1] = PR[GP1:90,1] + 2.748;
   1:  PR[GP1:91,2] = PR[GP1:90,2] + -47.081;
   1:  PR[GP1:91,3] = PR[GP1:90,3] + 118.645;
   1:L PR[91] 10mm/sec CNT100;
   1:  PR[GP1:91,1] = PR[GP1:90,1] + 5.987;
   1:  PR[GP1:91,2] = PR[GP1:90,2] + -46.726;
   1:L PR[91] 10mm/sec CNT100;
   1:  PR[GP1:91,1] = PR[GP1:90,1] + 19.618;
   1:  PR[GP1:91,2] = PR[GP1:90,2] + -44.178;
   1:L PR[91] 10mm/sec CNT100;
   1:  PR[GP1:91,1] = PR[GP1:90,1] + 22.670;
   1:  PR[GP1:91,2] = PR[GP1:90,2] + -42.785;
   1:L PR[91] 10mm/sec CNT100;
   1:  PR[GP1:91,1] = PR[GP1:90,1] + 34.304;
   1:  PR[GP1:91,2] = PR[GP1:90,2] + -35.579;
   1:L PR[91] 10mm/sec CNT100;
   1:  PR[GP1:91,1] = PR[GP1:90,1] + 36.823;
   1:  PR[GP1:91,2] = PR[GP1:90,2] + -33.238;
   1:L PR[91] 10mm/sec CNT100;
   1:  PR[GP1:91,1] = PR[GP1:90,1] + 43.298;
   1:  PR[GP1:91,2] = PR[GP1:90,2] + -25.437;
   1:L PR[91] 10mm/sec CNT100;
   1:  PR[GP1:91,1] = PR[GP1:90,1] + 44.977;
   1:  PR[GP1:91,2] = PR[GP1:90,2] + -22.348;
   1:L PR[91] 10mm/sec CNT100;
   1:  PR[GP1:91,1] = PR[GP1:90,1] + 49.038;
   1:  PR[GP1:91,2] = PR[GP1:90,2] + -13.149;
   1:L PR[91] 10mm/sec CNT100;
   1:  PR[GP1:91,1] = PR[GP1:90,1] + 49.619;
   1:  PR[GP1:91,2] = PR[GP1:90,2] + -9.695;
   1:L PR[91] 10mm/sec CNT100;
   1:  PR[GP1:91,1] = PR[GP1:90,1] + 49.620;
   1:  PR[GP1:91,2] = PR[GP1:90,2] + -9.614;
   1:L PR[91] 10mm/sec CNT100;
   1:  PR[GP1:91,1] = PR[GP1:90,1] + 50.998;
   1:  PR[GP1:91,2] = PR[GP1:90,2] + 0.271;
   1:L PR[91] 10mm/sec CNT100;
   1:  PR[GP1:91,1] = PR[GP1:90,1] + 50.425;
   1:  PR[GP1:91,2] = PR[GP1:90,2] + 3.738;
   1:L PR[91] 10mm/sec CNT100;
   1:  PR[GP1:91,1] = PR[GP1:90,1] + 49.032;
   1:  PR[GP1:91,2] = PR[GP1:90,2] + 13.722;
   1:L PR[91] 10mm/sec CNT100;
   1:  PR[GP1:91,1] = PR[GP1:90,1] + 44.975;
   1:  PR[GP1:91,2] = PR[GP1:90,2] + 22.913;
   1:L PR[91] 10mm/sec CNT100;
   1:  PR[GP1:91,1] = PR[GP1:90,1] + 43.289;
   1:  PR[GP1:91,2] = PR[GP1:90,2] + 26.007;
   1:L PR[91] 10mm/sec CNT100;
   1:  PR[GP1:91,1] = PR[GP1:90,1] + 36.813;
   1:  PR[GP1:91,2] = PR[GP1:90,2] + 33.808;
   1:L PR[91] 10mm/sec CNT100;
   1:  PR[GP1:91,1] = PR[GP1:90,1] + 34.286;
   1:  PR[GP1:91,2] = PR[GP1:90,2] + 36.149;
   1:L PR[91] 10mm/sec CNT100;
   1:  PR[GP1:91,1] = PR[GP1:90,1] + 22.651;
   1:  PR[GP1:91,2] = PR[GP1:90,2] + 43.355;
   1:L PR[91] 10mm/sec CNT100;
   1:  PR[GP1:91,1] = PR[GP1:90,1] + 19.591;
   1:  PR[GP1:91,2] = PR[GP1:90,2] + 44.743;
   1:L PR[91] 10mm/sec CNT100;
   1:  PR[GP1:91,1] = PR[GP1:90,1] + 5.959;
   1:  PR[GP1:91,2] = PR[GP1:90,2] + 47.291;
   1:L PR[91] 10mm/sec CNT100;
   1:  PR[GP1:91,1] = PR[GP1:90,1] + 2.717;
   1:  PR[GP1:91,2] = PR[GP1:90,2] + 47.637;
   1:L PR[91] 10mm/sec CNT100;
   1:  PR[GP1:91,1] = PR[GP1:90,1] + -0.265;
   1:  PR[GP1:91,2] = PR[GP1:90,2] + 47.113;
   1:L PR[91] 10mm/sec CNT100;
   1:  PR[GP1:91,1] = PR[GP1:90,1] + -3.249;
   1:  PR[GP1:91,2] = PR[GP1:90,2] + 47.637;
   1:L PR[91] 10mm/sec CNT100;
   1:  PR[GP1:91,1] = PR[GP1:90,1] + -6.491;
   1:  PR[GP1:91,2] = PR[GP1:90,2] + 47.292;
   1:L PR[91] 10mm/sec CNT100;
   1:  PR[GP1:91,1] = PR[GP1:90,1] + -20.120;
   1:  PR[GP1:91,2] = PR[GP1:90,2] + 44.743;
   1:L PR[91] 10mm/sec CNT100;
   1:  PR[GP1:91,1] = PR[GP1:90,1] + -23.180;
   1:  PR[GP1:91,2] = PR[GP1:90,2] + 43.353;
   1:L PR[91] 10mm/sec CNT100;
   1:  PR[GP1:91,1] = PR[GP1:90,1] + -34.811;
   1:  PR[GP1:91,2] = PR[GP1:90,2] + 36.149;
   1:L PR[91] 10mm/sec CNT100;
   1:  PR[GP1:91,1] = PR[GP1:90,1] + -37.339;
   1:  PR[GP1:91,2] = PR[GP1:90,2] + 33.811;
   1:L PR[91] 10mm/sec CNT100;
   1:  PR[GP1:91,1] = PR[GP1:90,1] + -43.815;
   1:  PR[GP1:91,2] = PR[GP1:90,2] + 26.010;
   1:L PR[91] 10mm/sec CNT100;
   1:  PR[GP1:91,1] = PR[GP1:90,1] + -45.501;
   1:  PR[GP1:91,2] = PR[GP1:90,2] + 22.910;
   1:L PR[91] 10mm/sec CNT100;
   1:  PR[GP1:91,1] = PR[GP1:90,1] + -49.562;
   1:  PR[GP1:91,2] = PR[GP1:90,2] + 13.711;
   1:L PR[91] 10mm/sec CNT100;
   1:  PR[GP1:91,1] = PR[GP1:90,1] + -50.145;
   1:  PR[GP1:91,2] = PR[GP1:90,2] + 10.254;
   1:L PR[91] 10mm/sec CNT100;
   1:  PR[GP1:91,1] = PR[GP1:90,1] + -50.146;
   1:  PR[GP1:91,2] = PR[GP1:90,2] + 10.173;
   1:L PR[91] 10mm/sec CNT100;
   1:  PR[GP1:91,1] = PR[GP1:90,1] + -51.525;
   1:  PR[GP1:91,2] = PR[GP1:90,2] + 0.287;
   1:L PR[91] 10mm/sec CNT100;
   1:  PR[GP1:91,1] = PR[GP1:90,1] + -50.954;
   1:  PR[GP1:91,2] = PR[GP1:90,2] + -3.169;
   1:L PR[91] 10mm/sec CNT100;
   1:  PR[GP1:91,1] = PR[GP1:90,1] + -49.561;
   1:  PR[GP1:91,2] = PR[GP1:90,2] + -13.153;
   1:L PR[91] 10mm/sec CNT100;
   1:  PR[GP1:91,1] = PR[GP1:90,1] + -45.503;
   1:  PR[GP1:91,2] = PR[GP1:90,2] + -22.345;
   1:L PR[91] 10mm/sec CNT100;
   1:  PR[GP1:91,1] = PR[GP1:90,1] + -43.824;
   1:  PR[GP1:91,2] = PR[GP1:90,2] + -25.440;
   1:L PR[91] 10mm/sec CNT100;
   1:  PR[GP1:91,1] = PR[GP1:90,1] + -37.348;
   1:  PR[GP1:91,2] = PR[GP1:90,2] + -33.241;
   1:L PR[91] 10mm/sec CNT100;
   1:  PR[GP1:91,1] = PR[GP1:90,1] + -34.829;
   1:  PR[GP1:91,2] = PR[GP1:90,2] + -35.579;
   1:L PR[91] 10mm/sec CNT100;
   1:  PR[GP1:91,1] = PR[GP1:90,1] + -23.199;
   1:  PR[GP1:91,2] = PR[GP1:90,2] + -42.783;
   1:L PR[91] 10mm/sec CNT100;
   1:  PR[GP1:91,1] = PR[GP1:90,1] + -20.147;
   1:  PR[GP1:91,2] = PR[GP1:90,2] + -44.177;
   1:L PR[91] 10mm/sec CNT100;
   1:  PR[GP1:91,1] = PR[GP1:90,1] + -6.520;
   1:  PR[GP1:91,2] = PR[GP1:90,2] + -46.726;
   1:L PR[91] 10mm/sec CNT100;
   1:  PR[GP1:91,1] = PR[GP1:90,1] + -3.281;
   1:  PR[GP1:91,2] = PR[GP1:90,2] + -47.081;
   1:L PR[91] 10mm/sec CNT100;
   1:  PR[GP1:91,1] = PR[GP1:90,1] + -0.265;
   1:  PR[GP1:91,2] = PR[GP1:90,2] + -46.576;
   1:L PR[91] 10mm/sec CNT100;
   1:  PR[GP1:91,1] = PR[GP1:90,1] + 2.559;
   1:  PR[GP1:91,2] = PR[GP1:90,2] + -47.210;
   1:  PR[GP1:91,3] = PR[GP1:90,3] + 119.255;
   1:L PR[91] 10mm/sec CNT100;
   1:  PR[GP1:91,1] = PR[GP1:90,1] + 5.586;
   1:  PR[GP1:91,2] = PR[GP1:90,2] + -46.877;
   1:L PR[91] 10mm/sec CNT100;
   1:  PR[GP1:91,1] = PR[GP1:90,1] + 19.492;
   1:  PR[GP1:91,2] = PR[GP1:90,2] + -44.278;
   1:L PR[91] 10mm/sec CNT100;
   1:  PR[GP1:91,1] = PR[GP1:90,1] + 22.345;
   1:  PR[GP1:91,2] = PR[GP1:90,2] + -42.976;
   1:L PR[91] 10mm/sec CNT100;
   1:  PR[GP1:91,1] = PR[GP1:90,1] + 34.225;
   1:  PR[GP1:91,2] = PR[GP1:90,2] + -35.618;
   1:L PR[91] 10mm/sec CNT100;
   1:  PR[GP1:91,1] = PR[GP1:90,1] + 36.581;
   1:  PR[GP1:91,2] = PR[GP1:90,2] + -33.428;
   1:L PR[91] 10mm/sec CNT100;
   1:  PR[GP1:91,1] = PR[GP1:90,1] + 43.201;
   1:  PR[GP1:91,2] = PR[GP1:90,2] + -25.454;
   1:L PR[91] 10mm/sec CNT100;
   1:  PR[GP1:91,1] = PR[GP1:90,1] + 44.771;
   1:  PR[GP1:91,2] = PR[GP1:90,2] + -22.564;
   1:L PR[91] 10mm/sec CNT100;
   1:  PR[GP1:91,1] = PR[GP1:90,1] + 48.925;
   1:  PR[GP1:91,2] = PR[GP1:90,2] + -13.154;
   1:L PR[91] 10mm/sec CNT100;
   1:  PR[GP1:91,1] = PR[GP1:90,1] + 49.468;
   1:  PR[GP1:91,2] = PR[GP1:90,2] + -9.926;
   1:L PR[91] 10mm/sec CNT100;
   1:  PR[GP1:91,1] = PR[GP1:90,1] + 49.469;
   1:  PR[GP1:91,2] = PR[GP1:90,2] + -9.851;
   1:L PR[91] 10mm/sec CNT100;
   1:  PR[GP1:91,1] = PR[GP1:90,1] + 50.880;
   1:  PR[GP1:91,2] = PR[GP1:90,2] + 0.271;
   1:L PR[91] 10mm/sec CNT100;
   1:  PR[GP1:91,1] = PR[GP1:90,1] + 50.344;
   1:  PR[GP1:91,2] = PR[GP1:90,2] + 3.514;
   1:L PR[91] 10mm/sec CNT100;
   1:  PR[GP1:91,1] = PR[GP1:90,1] + 48.920;
   1:  PR[GP1:91,2] = PR[GP1:90,2] + 13.726;
   1:L PR[91] 10mm/sec CNT100;
   1:  PR[GP1:91,1] = PR[GP1:90,1] + 44.769;
   1:  PR[GP1:91,2] = PR[GP1:90,2] + 23.129;
   1:L PR[91] 10mm/sec CNT100;
   1:  PR[GP1:91,1] = PR[GP1:90,1] + 43.192;
   1:  PR[GP1:91,2] = PR[GP1:90,2] + 26.023;
   1:L PR[91] 10mm/sec CNT100;
   1:  PR[GP1:91,1] = PR[GP1:90,1] + 36.572;
   1:  PR[GP1:91,2] = PR[GP1:90,2] + 33.997;
   1:L PR[91] 10mm/sec CNT100;
   1:  PR[GP1:91,1] = PR[GP1:90,1] + 34.208;
   1:  PR[GP1:91,2] = PR[GP1:90,2] + 36.187;
   1:L PR[91] 10mm/sec CNT100;
   1:  PR[GP1:91,1] = PR[GP1:90,1] + 22.327;
   1:  PR[GP1:91,2] = PR[GP1:90,2] + 43.545;
   1:L PR[91] 10mm/sec CNT100;
   1:  PR[GP1:91,1] = PR[GP1:90,1] + 19.466;
   1:  PR[GP1:91,2] = PR[GP1:90,2] + 44.843;
   1:L PR[91] 10mm/sec CNT100;
   1:  PR[GP1:91,1] = PR[GP1:90,1] + 5.560;
   1:  PR[GP1:91,2] = PR[GP1:90,2] + 47.442;
   1:L PR[91] 10mm/sec CNT100;
   1:  PR[GP1:91,1] = PR[GP1:90,1] + 2.530;
   1:  PR[GP1:91,2] = PR[GP1:90,2] + 47.766;
   1:L PR[91] 10mm/sec CNT100;
   1:  PR[GP1:91,1] = PR[GP1:90,1] + -0.265;
   1:  PR[GP1:91,2] = PR[GP1:90,2] + 47.274;
   1:L PR[91] 10mm/sec CNT100;
   1:  PR[GP1:91,1] = PR[GP1:90,1] + -3.062;
   1:  PR[GP1:91,2] = PR[GP1:90,2] + 47.766;
   1:L PR[91] 10mm/sec CNT100;
   1:  PR[GP1:91,1] = PR[GP1:90,1] + -6.093;
   1:  PR[GP1:91,2] = PR[GP1:90,2] + 47.443;
   1:L PR[91] 10mm/sec CNT100;
   1:  PR[GP1:91,1] = PR[GP1:90,1] + -19.995;
   1:  PR[GP1:91,2] = PR[GP1:90,2] + 44.842;
   1:L PR[91] 10mm/sec CNT100;
   1:  PR[GP1:91,1] = PR[GP1:90,1] + -22.856;
   1:  PR[GP1:91,2] = PR[GP1:90,2] + 43.544;
   1:L PR[91] 10mm/sec CNT100;
   1:  PR[GP1:91,1] = PR[GP1:90,1] + -34.734;
   1:  PR[GP1:91,2] = PR[GP1:90,2] + 36.187;
   1:L PR[91] 10mm/sec CNT100;
   1:  PR[GP1:91,1] = PR[GP1:90,1] + -37.097;
   1:  PR[GP1:91,2] = PR[GP1:90,2] + 34.000;
   1:L PR[91] 10mm/sec CNT100;
   1:  PR[GP1:91,1] = PR[GP1:90,1] + -43.718;
   1:  PR[GP1:91,2] = PR[GP1:90,2] + 26.025;
   1:L PR[91] 10mm/sec CNT100;
   1:  PR[GP1:91,1] = PR[GP1:90,1] + -45.295;
   1:  PR[GP1:91,2] = PR[GP1:90,2] + 23.126;
   1:L PR[91] 10mm/sec CNT100;
   1:  PR[GP1:91,1] = PR[GP1:90,1] + -49.449;
   1:  PR[GP1:91,2] = PR[GP1:90,2] + 13.715;
   1:L PR[91] 10mm/sec CNT100;
   1:  PR[GP1:91,1] = PR[GP1:90,1] + -49.994;
   1:  PR[GP1:91,2] = PR[GP1:90,2] + 10.484;
   1:L PR[91] 10mm/sec CNT100;
   1:  PR[GP1:91,1] = PR[GP1:90,1] + -49.995;
   1:  PR[GP1:91,2] = PR[GP1:90,2] + 10.409;
   1:L PR[91] 10mm/sec CNT100;
   1:  PR[GP1:91,1] = PR[GP1:90,1] + -51.407;
   1:  PR[GP1:91,2] = PR[GP1:90,2] + 0.287;
   1:L PR[91] 10mm/sec CNT100;
   1:  PR[GP1:91,1] = PR[GP1:90,1] + -50.873;
   1:  PR[GP1:91,2] = PR[GP1:90,2] + -2.946;
   1:L PR[91] 10mm/sec CNT100;
   1:  PR[GP1:91,1] = PR[GP1:90,1] + -49.448;
   1:  PR[GP1:91,2] = PR[GP1:90,2] + -13.158;
   1:L PR[91] 10mm/sec CNT100;
   1:  PR[GP1:91,1] = PR[GP1:90,1] + -45.297;
   1:  PR[GP1:91,2] = PR[GP1:90,2] + -22.562;
   1:L PR[91] 10mm/sec CNT100;
   1:  PR[GP1:91,1] = PR[GP1:90,1] + -43.727;
   1:  PR[GP1:91,2] = PR[GP1:90,2] + -25.456;
   1:L PR[91] 10mm/sec CNT100;
   1:  PR[GP1:91,1] = PR[GP1:90,1] + -37.106;
   1:  PR[GP1:91,2] = PR[GP1:90,2] + -33.431;
   1:L PR[91] 10mm/sec CNT100;
   1:  PR[GP1:91,1] = PR[GP1:90,1] + -34.751;
   1:  PR[GP1:91,2] = PR[GP1:90,2] + -35.618;
   1:L PR[91] 10mm/sec CNT100;
   1:  PR[GP1:91,1] = PR[GP1:90,1] + -22.873;
   1:  PR[GP1:91,2] = PR[GP1:90,2] + -42.974;
   1:L PR[91] 10mm/sec CNT100;
   1:  PR[GP1:91,1] = PR[GP1:90,1] + -20.020;
   1:  PR[GP1:91,2] = PR[GP1:90,2] + -44.277;
   1:L PR[91] 10mm/sec CNT100;
   1:  PR[GP1:91,1] = PR[GP1:90,1] + -6.119;
   1:  PR[GP1:91,2] = PR[GP1:90,2] + -46.877;
   1:L PR[91] 10mm/sec CNT100;
   1:  PR[GP1:91,1] = PR[GP1:90,1] + -3.092;
   1:  PR[GP1:91,2] = PR[GP1:90,2] + -47.210;
   1:L PR[91] 10mm/sec CNT100;
   1:  PR[GP1:91,1] = PR[GP1:90,1] + -0.265;
   1:  PR[GP1:91,2] = PR[GP1:90,2] + -46.736;
   1:L PR[91] 10mm/sec CNT100;
   1:  PR[GP1:91,1] = PR[GP1:90,1] + 2.370;
   1:  PR[GP1:91,2] = PR[GP1:90,2] + -47.338;
   1:  PR[GP1:91,3] = PR[GP1:90,3] + 119.865;
   1:L PR[91] 10mm/sec CNT100;
   1:  PR[GP1:91,1] = PR[GP1:90,1] + 5.186;
   1:  PR[GP1:91,2] = PR[GP1:90,2] + -47.029;
   1:L PR[91] 10mm/sec CNT100;
   1:  PR[GP1:91,1] = PR[GP1:90,1] + 19.365;
   1:  PR[GP1:91,2] = PR[GP1:90,2] + -44.378;
   1:L PR[91] 10mm/sec CNT100;
   1:  PR[GP1:91,1] = PR[GP1:90,1] + 22.019;
   1:  PR[GP1:91,2] = PR[GP1:90,2] + -43.167;
   1:L PR[91] 10mm/sec CNT100;
   1:  PR[GP1:91,1] = PR[GP1:90,1] + 34.147;
   1:  PR[GP1:91,2] = PR[GP1:90,2] + -35.656;
   1:L PR[91] 10mm/sec CNT100;
   1:  PR[GP1:91,1] = PR[GP1:90,1] + 36.339;
   1:  PR[GP1:91,2] = PR[GP1:90,2] + -33.618;
   1:L PR[91] 10mm/sec CNT100;
   1:  PR[GP1:91,1] = PR[GP1:90,1] + 43.103;
   1:  PR[GP1:91,2] = PR[GP1:90,2] + -25.470;
   1:L PR[91] 10mm/sec CNT100;
   1:  PR[GP1:91,1] = PR[GP1:90,1] + 44.565;
   1:  PR[GP1:91,2] = PR[GP1:90,2] + -22.781;
   1:L PR[91] 10mm/sec CNT100;
   1:  PR[GP1:91,1] = PR[GP1:90,1] + 48.812;
   1:  PR[GP1:91,2] = PR[GP1:90,2] + -13.159;
   1:L PR[91] 10mm/sec CNT100;
   1:  PR[GP1:91,1] = PR[GP1:90,1] + 49.323;
   1:  PR[GP1:91,2] = PR[GP1:90,2] + -10.119;
   1:L PR[91] 10mm/sec CNT100;
   1:  PR[GP1:91,1] = PR[GP1:90,1] + 50.762;
   1:  PR[GP1:91,2] = PR[GP1:90,2] + 0.271;
   1:L PR[91] 10mm/sec CNT100;
   1:  PR[GP1:91,1] = PR[GP1:90,1] + 50.263;
   1:  PR[GP1:91,2] = PR[GP1:90,2] + 3.290;
   1:L PR[91] 10mm/sec CNT100;
   1:  PR[GP1:91,1] = PR[GP1:90,1] + 48.807;
   1:  PR[GP1:91,2] = PR[GP1:90,2] + 13.731;
   1:L PR[91] 10mm/sec CNT100;
   1:  PR[GP1:91,1] = PR[GP1:90,1] + 44.563;
   1:  PR[GP1:91,2] = PR[GP1:90,2] + 23.345;
   1:L PR[91] 10mm/sec CNT100;
   1:  PR[GP1:91,1] = PR[GP1:90,1] + 43.095;
   1:  PR[GP1:91,2] = PR[GP1:90,2] + 26.038;
   1:L PR[91] 10mm/sec CNT100;
   1:  PR[GP1:91,1] = PR[GP1:90,1] + 36.331;
   1:  PR[GP1:91,2] = PR[GP1:90,2] + 34.187;
   1:L PR[91] 10mm/sec CNT100;
   1:  PR[GP1:91,1] = PR[GP1:90,1] + 34.131;
   1:  PR[GP1:91,2] = PR[GP1:90,2] + 36.224;
   1:L PR[91] 10mm/sec CNT100;
   1:  PR[GP1:91,1] = PR[GP1:90,1] + 22.003;
   1:  PR[GP1:91,2] = PR[GP1:90,2] + 43.736;
   1:L PR[91] 10mm/sec CNT100;
   1:  PR[GP1:91,1] = PR[GP1:90,1] + 19.342;
   1:  PR[GP1:91,2] = PR[GP1:90,2] + 44.943;
   1:L PR[91] 10mm/sec CNT100;
   1:  PR[GP1:91,1] = PR[GP1:90,1] + 5.161;
   1:  PR[GP1:91,2] = PR[GP1:90,2] + 47.594;
   1:L PR[91] 10mm/sec CNT100;
   1:  PR[GP1:91,1] = PR[GP1:90,1] + 2.343;
   1:  PR[GP1:91,2] = PR[GP1:90,2] + 47.895;
   1:L PR[91] 10mm/sec CNT100;
   1:  PR[GP1:91,1] = PR[GP1:90,1] + -0.265;
   1:  PR[GP1:91,2] = PR[GP1:90,2] + 47.436;
   1:L PR[91] 10mm/sec CNT100;
   1:  PR[GP1:91,1] = PR[GP1:90,1] + -2.875;
   1:  PR[GP1:91,2] = PR[GP1:90,2] + 47.894;
   1:L PR[91] 10mm/sec CNT100;
   1:  PR[GP1:91,1] = PR[GP1:90,1] + -5.694;
   1:  PR[GP1:91,2] = PR[GP1:90,2] + 47.594;
   1:L PR[91] 10mm/sec CNT100;
   1:  PR[GP1:91,1] = PR[GP1:90,1] + -19.871;
   1:  PR[GP1:91,2] = PR[GP1:90,2] + 44.942;
   1:L PR[91] 10mm/sec CNT100;
   1:  PR[GP1:91,1] = PR[GP1:90,1] + -22.532;
   1:  PR[GP1:91,2] = PR[GP1:90,2] + 43.734;
   1:L PR[91] 10mm/sec CNT100;
   1:  PR[GP1:91,1] = PR[GP1:90,1] + -34.657;
   1:  PR[GP1:91,2] = PR[GP1:90,2] + 36.225;
   1:L PR[91] 10mm/sec CNT100;
   1:  PR[GP1:91,1] = PR[GP1:90,1] + -36.856;
   1:  PR[GP1:91,2] = PR[GP1:90,2] + 34.190;
   1:L PR[91] 10mm/sec CNT100;
   1:  PR[GP1:91,1] = PR[GP1:90,1] + -43.621;
   1:  PR[GP1:91,2] = PR[GP1:90,2] + 26.041;
   1:L PR[91] 10mm/sec CNT100;
   1:  PR[GP1:91,1] = PR[GP1:90,1] + -45.088;
   1:  PR[GP1:91,2] = PR[GP1:90,2] + 23.343;
   1:L PR[91] 10mm/sec CNT100;
   1:  PR[GP1:91,1] = PR[GP1:90,1] + -49.336;
   1:  PR[GP1:91,2] = PR[GP1:90,2] + 13.720;
   1:L PR[91] 10mm/sec CNT100;
   1:  PR[GP1:91,1] = PR[GP1:90,1] + -49.843;
   1:  PR[GP1:91,2] = PR[GP1:90,2] + 10.715;
   1:L PR[91] 10mm/sec CNT100;
   1:  PR[GP1:91,1] = PR[GP1:90,1] + -49.844;
   1:  PR[GP1:91,2] = PR[GP1:90,2] + 10.646;
   1:L PR[91] 10mm/sec CNT100;
   1:  PR[GP1:91,1] = PR[GP1:90,1] + -51.289;
   1:  PR[GP1:91,2] = PR[GP1:90,2] + 0.287;
   1:L PR[91] 10mm/sec CNT100;
   1:  PR[GP1:91,1] = PR[GP1:90,1] + -50.792;
   1:  PR[GP1:91,2] = PR[GP1:90,2] + -2.722;
   1:L PR[91] 10mm/sec CNT100;
   1:  PR[GP1:91,1] = PR[GP1:90,1] + -49.335;
   1:  PR[GP1:91,2] = PR[GP1:90,2] + -13.164;
   1:L PR[91] 10mm/sec CNT100;
   1:  PR[GP1:91,1] = PR[GP1:90,1] + -45.091;
   1:  PR[GP1:91,2] = PR[GP1:90,2] + -22.778;
   1:L PR[91] 10mm/sec CNT100;
   1:  PR[GP1:91,1] = PR[GP1:90,1] + -43.629;
   1:  PR[GP1:91,2] = PR[GP1:90,2] + -25.473;
   1:L PR[91] 10mm/sec CNT100;
   1:  PR[GP1:91,1] = PR[GP1:90,1] + -36.864;
   1:  PR[GP1:91,2] = PR[GP1:90,2] + -33.621;
   1:L PR[91] 10mm/sec CNT100;
   1:  PR[GP1:91,1] = PR[GP1:90,1] + -34.672;
   1:  PR[GP1:91,2] = PR[GP1:90,2] + -35.656;
   1:L PR[91] 10mm/sec CNT100;
   1:  PR[GP1:91,1] = PR[GP1:90,1] + -22.548;
   1:  PR[GP1:91,2] = PR[GP1:90,2] + -43.165;
   1:L PR[91] 10mm/sec CNT100;
   1:  PR[GP1:91,1] = PR[GP1:90,1] + -19.894;
   1:  PR[GP1:91,2] = PR[GP1:90,2] + -44.378;
   1:L PR[91] 10mm/sec CNT100;
   1:  PR[GP1:91,1] = PR[GP1:90,1] + -5.719;
   1:  PR[GP1:91,2] = PR[GP1:90,2] + -47.029;
   1:L PR[91] 10mm/sec CNT100;
   1:  PR[GP1:91,1] = PR[GP1:90,1] + -2.903;
   1:  PR[GP1:91,2] = PR[GP1:90,2] + -47.338;
   1:L PR[91] 10mm/sec CNT100;
   1:  PR[GP1:91,1] = PR[GP1:90,1] + -0.265;
   1:  PR[GP1:91,2] = PR[GP1:90,2] + -46.896;
   1:L PR[91] 10mm/sec CNT100;
   1:  PR[GP1:91,1] = PR[GP1:90,1] + 2.180;
   1:  PR[GP1:91,2] = PR[GP1:90,2] + -47.467;
   1:  PR[GP1:91,3] = PR[GP1:90,3] + 120.475;
   1:L PR[91] 10mm/sec CNT100;
   1:  PR[GP1:91,1] = PR[GP1:90,1] + 4.785;
   1:  PR[GP1:91,2] = PR[GP1:90,2] + -47.180;
   1:L PR[91] 10mm/sec CNT100;
   1:  PR[GP1:91,1] = PR[GP1:90,1] + 19.239;
   1:  PR[GP1:91,2] = PR[GP1:90,2] + -44.479;
   1:L PR[91] 10mm/sec CNT100;
   1:  PR[GP1:91,1] = PR[GP1:90,1] + 21.694;
   1:  PR[GP1:91,2] = PR[GP1:90,2] + -43.358;
   1:L PR[91] 10mm/sec CNT100;
   1:  PR[GP1:91,1] = PR[GP1:90,1] + 34.069;
   1:  PR[GP1:91,2] = PR[GP1:90,2] + -35.694;
   1:L PR[91] 10mm/sec CNT100;
   1:  PR[GP1:91,1] = PR[GP1:90,1] + 36.097;
   1:  PR[GP1:91,2] = PR[GP1:90,2] + -33.809;
   1:L PR[91] 10mm/sec CNT100;
   1:  PR[GP1:91,1] = PR[GP1:90,1] + 43.005;
   1:  PR[GP1:91,2] = PR[GP1:90,2] + -25.487;
   1:L PR[91] 10mm/sec CNT100;
   1:  PR[GP1:91,1] = PR[GP1:90,1] + 44.359;
   1:  PR[GP1:91,2] = PR[GP1:90,2] + -22.997;
   1:L PR[91] 10mm/sec CNT100;
   1:  PR[GP1:91,1] = PR[GP1:90,1] + 48.699;
   1:  PR[GP1:91,2] = PR[GP1:90,2] + -13.164;
   1:L PR[91] 10mm/sec CNT100;
   1:  PR[GP1:91,1] = PR[GP1:90,1] + 49.172;
   1:  PR[GP1:91,2] = PR[GP1:90,2] + -10.350;
   1:L PR[91] 10mm/sec CNT100;
   1:  PR[GP1:91,1] = PR[GP1:90,1] + 50.644;
   1:  PR[GP1:91,2] = PR[GP1:90,2] + 0.271;
   1:L PR[91] 10mm/sec CNT100;
   1:  PR[GP1:91,1] = PR[GP1:90,1] + 50.182;
   1:  PR[GP1:91,2] = PR[GP1:90,2] + 3.066;
   1:L PR[91] 10mm/sec CNT100;
   1:  PR[GP1:91,1] = PR[GP1:90,1] + 48.694;
   1:  PR[GP1:91,2] = PR[GP1:90,2] + 13.736;
   1:L PR[91] 10mm/sec CNT100;
   1:  PR[GP1:91,1] = PR[GP1:90,1] + 44.357;
   1:  PR[GP1:91,2] = PR[GP1:90,2] + 23.561;
   1:L PR[91] 10mm/sec CNT100;
   1:  PR[GP1:91,1] = PR[GP1:90,1] + 42.998;
   1:  PR[GP1:91,2] = PR[GP1:90,2] + 26.054;
   1:L PR[91] 10mm/sec CNT100;
   1:  PR[GP1:91,1] = PR[GP1:90,1] + 36.090;
   1:  PR[GP1:91,2] = PR[GP1:90,2] + 34.376;
   1:L PR[91] 10mm/sec CNT100;
   1:  PR[GP1:91,1] = PR[GP1:90,1] + 34.054;
   1:  PR[GP1:91,2] = PR[GP1:90,2] + 36.262;
   1:L PR[91] 10mm/sec CNT100;
   1:  PR[GP1:91,1] = PR[GP1:90,1] + 21.679;
   1:  PR[GP1:91,2] = PR[GP1:90,2] + 43.926;
   1:L PR[91] 10mm/sec CNT100;
   1:  PR[GP1:91,1] = PR[GP1:90,1] + 19.217;
   1:  PR[GP1:91,2] = PR[GP1:90,2] + 45.043;
   1:L PR[91] 10mm/sec CNT100;
   1:  PR[GP1:91,1] = PR[GP1:90,1] + 4.763;
   1:  PR[GP1:91,2] = PR[GP1:90,2] + 47.745;
   1:L PR[91] 10mm/sec CNT100;
   1:  PR[GP1:91,1] = PR[GP1:90,1] + 2.155;
   1:  PR[GP1:91,2] = PR[GP1:90,2] + 48.023;
   1:L PR[91] 10mm/sec CNT100;
   1:  PR[GP1:91,1] = PR[GP1:90,1] + -0.265;
   1:  PR[GP1:91,2] = PR[GP1:90,2] + 47.597;
   1:L PR[91] 10mm/sec CNT100;
   1:  PR[GP1:91,1] = PR[GP1:90,1] + -2.688;
   1:  PR[GP1:91,2] = PR[GP1:90,2] + 48.023;
   1:L PR[91] 10mm/sec CNT100;
   1:  PR[GP1:91,1] = PR[GP1:90,1] + -5.296;
   1:  PR[GP1:91,2] = PR[GP1:90,2] + 47.745;
   1:L PR[91] 10mm/sec CNT100;
   1:  PR[GP1:91,1] = PR[GP1:90,1] + -19.746;
   1:  PR[GP1:91,2] = PR[GP1:90,2] + 45.042;
   1:L PR[91] 10mm/sec CNT100;
   1:  PR[GP1:91,1] = PR[GP1:90,1] + -22.207;
   1:  PR[GP1:91,2] = PR[GP1:90,2] + 43.925;
   1:L PR[91] 10mm/sec CNT100;
   1:  PR[GP1:91,1] = PR[GP1:90,1] + -34.579;
   1:  PR[GP1:91,2] = PR[GP1:90,2] + 36.262;
   1:L PR[91] 10mm/sec CNT100;
   1:  PR[GP1:91,1] = PR[GP1:90,1] + -36.615;
   1:  PR[GP1:91,2] = PR[GP1:90,2] + 34.379;
   1:L PR[91] 10mm/sec CNT100;
   1:  PR[GP1:91,1] = PR[GP1:90,1] + -43.524;
   1:  PR[GP1:91,2] = PR[GP1:90,2] + 26.057;
   1:L PR[91] 10mm/sec CNT100;
   1:  PR[GP1:91,1] = PR[GP1:90,1] + -44.882;
   1:  PR[GP1:91,2] = PR[GP1:90,2] + 23.559;
   1:L PR[91] 10mm/sec CNT100;
   1:  PR[GP1:91,1] = PR[GP1:90,1] + -49.224;
   1:  PR[GP1:91,2] = PR[GP1:90,2] + 13.725;
   1:L PR[91] 10mm/sec CNT100;
   1:  PR[GP1:91,1] = PR[GP1:90,1] + -49.692;
   1:  PR[GP1:91,2] = PR[GP1:90,2] + 10.946;
   1:L PR[91] 10mm/sec CNT100;
   1:  PR[GP1:91,1] = PR[GP1:90,1] + -49.693;
   1:  PR[GP1:91,2] = PR[GP1:90,2] + 10.882;
   1:L PR[91] 10mm/sec CNT100;
   1:  PR[GP1:91,1] = PR[GP1:90,1] + -51.171;
   1:  PR[GP1:91,2] = PR[GP1:90,2] + 0.287;
   1:L PR[91] 10mm/sec CNT100;
   1:  PR[GP1:91,1] = PR[GP1:90,1] + -50.711;
   1:  PR[GP1:91,2] = PR[GP1:90,2] + -2.499;
   1:L PR[91] 10mm/sec CNT100;
   1:  PR[GP1:91,1] = PR[GP1:90,1] + -49.222;
   1:  PR[GP1:91,2] = PR[GP1:90,2] + -13.169;
   1:L PR[91] 10mm/sec CNT100;
   1:  PR[GP1:91,1] = PR[GP1:90,1] + -44.884;
   1:  PR[GP1:91,2] = PR[GP1:90,2] + -22.995;
   1:L PR[91] 10mm/sec CNT100;
   1:  PR[GP1:91,1] = PR[GP1:90,1] + -43.531;
   1:  PR[GP1:91,2] = PR[GP1:90,2] + -25.489;
   1:L PR[91] 10mm/sec CNT100;
   1:  PR[GP1:91,1] = PR[GP1:90,1] + -36.622;
   1:  PR[GP1:91,2] = PR[GP1:90,2] + -33.811;
   1:L PR[91] 10mm/sec CNT100;
   1:  PR[GP1:91,1] = PR[GP1:90,1] + -34.594;
   1:  PR[GP1:91,2] = PR[GP1:90,2] + -35.694;
   1:L PR[91] 10mm/sec CNT100;
   1:  PR[GP1:91,1] = PR[GP1:90,1] + -22.223;
   1:  PR[GP1:91,2] = PR[GP1:90,2] + -43.357;
   1:L PR[91] 10mm/sec CNT100;
   1:  PR[GP1:91,1] = PR[GP1:90,1] + -19.768;
   1:  PR[GP1:91,2] = PR[GP1:90,2] + -44.478;
   1:L PR[91] 10mm/sec CNT100;
   1:  PR[GP1:91,1] = PR[GP1:90,1] + -5.319;
   1:  PR[GP1:91,2] = PR[GP1:90,2] + -47.181;
   1:L PR[91] 10mm/sec CNT100;
   1:  PR[GP1:91,1] = PR[GP1:90,1] + -2.713;
   1:  PR[GP1:91,2] = PR[GP1:90,2] + -47.467;
   1:L PR[91] 10mm/sec CNT100;
   1:  PR[GP1:91,1] = PR[GP1:90,1] + -0.265;
   1:  PR[GP1:91,2] = PR[GP1:90,2] + -47.056;
   1:L PR[91] 10mm/sec CNT100;
   1:  PR[GP1:91,1] = PR[GP1:90,1] + 1.991;
   1:  PR[GP1:91,2] = PR[GP1:90,2] + -47.595;
   1:  PR[GP1:91,3] = PR[GP1:90,3] + 121.085;
   1:L PR[91] 10mm/sec CNT100;
   1:  PR[GP1:91,1] = PR[GP1:90,1] + 4.385;
   1:  PR[GP1:91,2] = PR[GP1:90,2] + -47.332;
   1:L PR[91] 10mm/sec CNT100;
   1:  PR[GP1:91,1] = PR[GP1:90,1] + 19.113;
   1:  PR[GP1:91,2] = PR[GP1:90,2] + -44.579;
   1:L PR[91] 10mm/sec CNT100;
   1:  PR[GP1:91,1] = PR[GP1:90,1] + 21.368;
   1:  PR[GP1:91,2] = PR[GP1:90,2] + -43.550;
   1:L PR[91] 10mm/sec CNT100;
   1:  PR[GP1:91,1] = PR[GP1:90,1] + 33.990;
   1:  PR[GP1:91,2] = PR[GP1:90,2] + -35.733;
   1:L PR[91] 10mm/sec CNT100;
   1:  PR[GP1:91,1] = PR[GP1:90,1] + 35.855;
   1:  PR[GP1:91,2] = PR[GP1:90,2] + -33.999;
   1:L PR[91] 10mm/sec CNT100;
   1:  PR[GP1:91,1] = PR[GP1:90,1] + 42.908;
   1:  PR[GP1:91,2] = PR[GP1:90,2] + -25.503;
   1:L PR[91] 10mm/sec CNT100;
   1:  PR[GP1:91,1] = PR[GP1:90,1] + 44.152;
   1:  PR[GP1:91,2] = PR[GP1:90,2] + -23.213;
   1:L PR[91] 10mm/sec CNT100;
   1:  PR[GP1:91,1] = PR[GP1:90,1] + 48.586;
   1:  PR[GP1:91,2] = PR[GP1:90,2] + -13.169;
   1:L PR[91] 10mm/sec CNT100;
   1:  PR[GP1:91,1] = PR[GP1:90,1] + 49.021;
   1:  PR[GP1:91,2] = PR[GP1:90,2] + -10.581;
   1:L PR[91] 10mm/sec CNT100;
   1:  PR[GP1:91,1] = PR[GP1:90,1] + 50.527;
   1:  PR[GP1:91,2] = PR[GP1:90,2] + 0.271;
   1:L PR[91] 10mm/sec CNT100;
   1:  PR[GP1:91,1] = PR[GP1:90,1] + 50.101;
   1:  PR[GP1:91,2] = PR[GP1:90,2] + 2.842;
   1:L PR[91] 10mm/sec CNT100;
   1:  PR[GP1:91,1] = PR[GP1:90,1] + 48.581;
   1:  PR[GP1:91,2] = PR[GP1:90,2] + 13.740;
   1:L PR[91] 10mm/sec CNT100;
   1:  PR[GP1:91,1] = PR[GP1:90,1] + 44.151;
   1:  PR[GP1:91,2] = PR[GP1:90,2] + 23.776;
   1:L PR[91] 10mm/sec CNT100;
   1:  PR[GP1:91,1] = PR[GP1:90,1] + 42.901;
   1:  PR[GP1:91,2] = PR[GP1:90,2] + 26.070;
   1:L PR[91] 10mm/sec CNT100;
   1:  PR[GP1:91,1] = PR[GP1:90,1] + 35.848;
   1:  PR[GP1:91,2] = PR[GP1:90,2] + 34.566;
   1:L PR[91] 10mm/sec CNT100;
   1:  PR[GP1:91,1] = PR[GP1:90,1] + 33.977;
   1:  PR[GP1:91,2] = PR[GP1:90,2] + 36.299;
   1:L PR[91] 10mm/sec CNT100;
   1:  PR[GP1:91,1] = PR[GP1:90,1] + 21.355;
   1:  PR[GP1:91,2] = PR[GP1:90,2] + 44.117;
   1:L PR[91] 10mm/sec CNT100;
   1:  PR[GP1:91,1] = PR[GP1:90,1] + 19.093;
   1:  PR[GP1:91,2] = PR[GP1:90,2] + 45.143;
   1:L PR[91] 10mm/sec CNT100;
   1:  PR[GP1:91,1] = PR[GP1:90,1] + 4.364;
   1:  PR[GP1:91,2] = PR[GP1:90,2] + 47.896;
   1:L PR[91] 10mm/sec CNT100;
   1:  PR[GP1:91,1] = PR[GP1:90,1] + 1.968;
   1:  PR[GP1:91,2] = PR[GP1:90,2] + 48.152;
   1:L PR[91] 10mm/sec CNT100;
   1:  PR[GP1:91,1] = PR[GP1:90,1] + -0.265;
   1:  PR[GP1:91,2] = PR[GP1:90,2] + 47.759;
   1:L PR[91] 10mm/sec CNT100;
   1:  PR[GP1:91,1] = PR[GP1:90,1] + -2.501;
   1:  PR[GP1:91,2] = PR[GP1:90,2] + 48.152;
   1:L PR[91] 10mm/sec CNT100;
   1:  PR[GP1:91,1] = PR[GP1:90,1] + -4.897;
   1:  PR[GP1:91,2] = PR[GP1:90,2] + 47.896;
   1:L PR[91] 10mm/sec CNT100;
   1:  PR[GP1:91,1] = PR[GP1:90,1] + -19.622;
   1:  PR[GP1:91,2] = PR[GP1:90,2] + 45.142;
   1:L PR[91] 10mm/sec CNT100;
   1:  PR[GP1:91,1] = PR[GP1:90,1] + -21.883;
   1:  PR[GP1:91,2] = PR[GP1:90,2] + 44.115;
   1:L PR[91] 10mm/sec CNT100;
   1:  PR[GP1:91,1] = PR[GP1:90,1] + -34.502;
   1:  PR[GP1:91,2] = PR[GP1:90,2] + 36.300;
   1:L PR[91] 10mm/sec CNT100;
   1:  PR[GP1:91,1] = PR[GP1:90,1] + -36.373;
   1:  PR[GP1:91,2] = PR[GP1:90,2] + 34.569;
   1:L PR[91] 10mm/sec CNT100;
   1:  PR[GP1:91,1] = PR[GP1:90,1] + -43.427;
   1:  PR[GP1:91,2] = PR[GP1:90,2] + 26.073;
   1:L PR[91] 10mm/sec CNT100;
   1:  PR[GP1:91,1] = PR[GP1:90,1] + -44.676;
   1:  PR[GP1:91,2] = PR[GP1:90,2] + 23.775;
   1:L PR[91] 10mm/sec CNT100;
   1:  PR[GP1:91,1] = PR[GP1:90,1] + -49.111;
   1:  PR[GP1:91,2] = PR[GP1:90,2] + 13.730;
   1:L PR[91] 10mm/sec CNT100;
   1:  PR[GP1:91,1] = PR[GP1:90,1] + -49.541;
   1:  PR[GP1:91,2] = PR[GP1:90,2] + 11.177;
   1:L PR[91] 10mm/sec CNT100;
   1:  PR[GP1:91,1] = PR[GP1:90,1] + -49.542;
   1:  PR[GP1:91,2] = PR[GP1:90,2] + 11.118;
   1:L PR[91] 10mm/sec CNT100;
   1:  PR[GP1:91,1] = PR[GP1:90,1] + -51.053;
   1:  PR[GP1:91,2] = PR[GP1:90,2] + 0.287;
   1:L PR[91] 10mm/sec CNT100;
   1:  PR[GP1:91,1] = PR[GP1:90,1] + -50.629;
   1:  PR[GP1:91,2] = PR[GP1:90,2] + -2.275;
   1:L PR[91] 10mm/sec CNT100;
   1:  PR[GP1:91,1] = PR[GP1:90,1] + -49.109;
   1:  PR[GP1:91,2] = PR[GP1:90,2] + -13.174;
   1:L PR[91] 10mm/sec CNT100;
   1:  PR[GP1:91,1] = PR[GP1:90,1] + -44.678;
   1:  PR[GP1:91,2] = PR[GP1:90,2] + -23.211;
   1:L PR[91] 10mm/sec CNT100;
   1:  PR[GP1:91,1] = PR[GP1:90,1] + -43.433;
   1:  PR[GP1:91,2] = PR[GP1:90,2] + -25.506;
   1:L PR[91] 10mm/sec CNT100;
   1:  PR[GP1:91,1] = PR[GP1:90,1] + -36.380;
   1:  PR[GP1:91,2] = PR[GP1:90,2] + -34.002;
   1:L PR[91] 10mm/sec CNT100;
   1:  PR[GP1:91,1] = PR[GP1:90,1] + -34.516;
   1:  PR[GP1:91,2] = PR[GP1:90,2] + -35.733;
   1:L PR[91] 10mm/sec CNT100;
   1:  PR[GP1:91,1] = PR[GP1:90,1] + -21.897;
   1:  PR[GP1:91,2] = PR[GP1:90,2] + -43.548;
   1:L PR[91] 10mm/sec CNT100;
   1:  PR[GP1:91,1] = PR[GP1:90,1] + -19.642;
   1:  PR[GP1:91,2] = PR[GP1:90,2] + -44.578;
   1:L PR[91] 10mm/sec CNT100;
   1:  PR[GP1:91,1] = PR[GP1:90,1] + -4.918;
   1:  PR[GP1:91,2] = PR[GP1:90,2] + -47.332;
   1:L PR[91] 10mm/sec CNT100;
   1:  PR[GP1:91,1] = PR[GP1:90,1] + -2.524;
   1:  PR[GP1:91,2] = PR[GP1:90,2] + -47.595;
   1:L PR[91] 10mm/sec CNT100;
   1:  PR[GP1:91,1] = PR[GP1:90,1] + -0.265;
   1:  PR[GP1:91,2] = PR[GP1:90,2] + -47.216;
   1:L PR[91] 10mm/sec CNT100;
   1:  PR[GP1:91,1] = PR[GP1:90,1] + 1.802;
   1:  PR[GP1:91,2] = PR[GP1:90,2] + -47.724;
   1:  PR[GP1:91,3] = PR[GP1:90,3] + 121.695;
   1:L PR[91] 10mm/sec CNT100;
   1:  PR[GP1:91,1] = PR[GP1:90,1] + 3.984;
   1:  PR[GP1:91,2] = PR[GP1:90,2] + -47.484;
   1:L PR[91] 10mm/sec CNT100;
   1:  PR[GP1:91,1] = PR[GP1:90,1] + 18.987;
   1:  PR[GP1:91,2] = PR[GP1:90,2] + -44.680;
   1:L PR[91] 10mm/sec CNT100;
   1:  PR[GP1:91,1] = PR[GP1:90,1] + 21.043;
   1:  PR[GP1:91,2] = PR[GP1:90,2] + -43.741;
   1:L PR[91] 10mm/sec CNT100;
   1:  PR[GP1:91,1] = PR[GP1:90,1] + 33.912;
   1:  PR[GP1:91,2] = PR[GP1:90,2] + -35.771;
   1:L PR[91] 10mm/sec CNT100;
   1:  PR[GP1:91,1] = PR[GP1:90,1] + 35.613;
   1:  PR[GP1:91,2] = PR[GP1:90,2] + -34.189;
   1:L PR[91] 10mm/sec CNT100;
   1:  PR[GP1:91,1] = PR[GP1:90,1] + 42.810;
   1:  PR[GP1:91,2] = PR[GP1:90,2] + -25.520;
   1:L PR[91] 10mm/sec CNT100;
   1:  PR[GP1:91,1] = PR[GP1:90,1] + 43.946;
   1:  PR[GP1:91,2] = PR[GP1:90,2] + -23.429;
   1:L PR[91] 10mm/sec CNT100;
   1:  PR[GP1:91,1] = PR[GP1:90,1] + 48.473;
   1:  PR[GP1:91,2] = PR[GP1:90,2] + -13.174;
   1:L PR[91] 10mm/sec CNT100;
   1:  PR[GP1:91,1] = PR[GP1:90,1] + 48.871;
   1:  PR[GP1:91,2] = PR[GP1:90,2] + -10.811;
   1:L PR[91] 10mm/sec CNT100;
   1:  PR[GP1:91,1] = PR[GP1:90,1] + 50.409;
   1:  PR[GP1:91,2] = PR[GP1:90,2] + 0.271;
   1:L PR[91] 10mm/sec CNT100;
   1:  PR[GP1:91,1] = PR[GP1:90,1] + 50.020;
   1:  PR[GP1:91,2] = PR[GP1:90,2] + 2.617;
   1:L PR[91] 10mm/sec CNT100;
   1:  PR[GP1:91,1] = PR[GP1:90,1] + 48.468;
   1:  PR[GP1:91,2] = PR[GP1:90,2] + 13.745;
   1:L PR[91] 10mm/sec CNT100;
   1:  PR[GP1:91,1] = PR[GP1:90,1] + 43.944;
   1:  PR[GP1:91,2] = PR[GP1:90,2] + 23.992;
   1:L PR[91] 10mm/sec CNT100;
   1:  PR[GP1:91,1] = PR[GP1:90,1] + 42.804;
   1:  PR[GP1:91,2] = PR[GP1:90,2] + 26.086;
   1:L PR[91] 10mm/sec CNT100;
   1:  PR[GP1:91,1] = PR[GP1:90,1] + 35.607;
   1:  PR[GP1:91,2] = PR[GP1:90,2] + 34.755;
   1:L PR[91] 10mm/sec CNT100;
   1:  PR[GP1:91,1] = PR[GP1:90,1] + 33.900;
   1:  PR[GP1:91,2] = PR[GP1:90,2] + 36.337;
   1:L PR[91] 10mm/sec CNT100;
   1:  PR[GP1:91,1] = PR[GP1:90,1] + 21.030;
   1:  PR[GP1:91,2] = PR[GP1:90,2] + 44.307;
   1:L PR[91] 10mm/sec CNT100;
   1:  PR[GP1:91,1] = PR[GP1:90,1] + 18.968;
   1:  PR[GP1:91,2] = PR[GP1:90,2] + 45.243;
   1:L PR[91] 10mm/sec CNT100;
   1:  PR[GP1:91,1] = PR[GP1:90,1] + 3.965;
   1:  PR[GP1:91,2] = PR[GP1:90,2] + 48.047;
   1:L PR[91] 10mm/sec CNT100;
   1:  PR[GP1:91,1] = PR[GP1:90,1] + 1.781;
   1:  PR[GP1:91,2] = PR[GP1:90,2] + 48.280;
   1:L PR[91] 10mm/sec CNT100;
   1:  PR[GP1:91,1] = PR[GP1:90,1] + -0.265;
   1:  PR[GP1:91,2] = PR[GP1:90,2] + 47.920;
   1:L PR[91] 10mm/sec CNT100;
   1:  PR[GP1:91,1] = PR[GP1:90,1] + -2.314;
   1:  PR[GP1:91,2] = PR[GP1:90,2] + 48.280;
   1:L PR[91] 10mm/sec CNT100;
   1:  PR[GP1:91,1] = PR[GP1:90,1] + -4.499;
   1:  PR[GP1:91,2] = PR[GP1:90,2] + 48.047;
   1:L PR[91] 10mm/sec CNT100;
   1:  PR[GP1:91,1] = PR[GP1:90,1] + -19.497;
   1:  PR[GP1:91,2] = PR[GP1:90,2] + 45.242;
   1:L PR[91] 10mm/sec CNT100;
   1:  PR[GP1:91,1] = PR[GP1:90,1] + -21.559;
   1:  PR[GP1:91,2] = PR[GP1:90,2] + 44.306;
   1:L PR[91] 10mm/sec CNT100;
   1:  PR[GP1:91,1] = PR[GP1:90,1] + -34.425;
   1:  PR[GP1:91,2] = PR[GP1:90,2] + 36.337;
   1:L PR[91] 10mm/sec CNT100;
   1:  PR[GP1:91,1] = PR[GP1:90,1] + -36.132;
   1:  PR[GP1:91,2] = PR[GP1:90,2] + 34.758;
   1:L PR[91] 10mm/sec CNT100;
   1:  PR[GP1:91,1] = PR[GP1:90,1] + -43.330;
   1:  PR[GP1:91,2] = PR[GP1:90,2] + 26.088;
   1:L PR[91] 10mm/sec CNT100;
   1:  PR[GP1:91,1] = PR[GP1:90,1] + -44.470;
   1:  PR[GP1:91,2] = PR[GP1:90,2] + 23.991;
   1:L PR[91] 10mm/sec CNT100;
   1:  PR[GP1:91,1] = PR[GP1:90,1] + -48.998;
   1:  PR[GP1:91,2] = PR[GP1:90,2] + 13.736;
   1:L PR[91] 10mm/sec CNT100;
   1:  PR[GP1:91,1] = PR[GP1:90,1] + -49.397;
   1:  PR[GP1:91,2] = PR[GP1:90,2] + 11.309;
   1:L PR[91] 10mm/sec CNT100;
   1:  PR[GP1:91,1] = PR[GP1:90,1] + -50.935;
   1:  PR[GP1:91,2] = PR[GP1:90,2] + 0.287;
   1:L PR[91] 10mm/sec CNT100;
   1:  PR[GP1:91,1] = PR[GP1:90,1] + -50.548;
   1:  PR[GP1:91,2] = PR[GP1:90,2] + -2.052;
   1:L PR[91] 10mm/sec CNT100;
   1:  PR[GP1:91,1] = PR[GP1:90,1] + -48.996;
   1:  PR[GP1:91,2] = PR[GP1:90,2] + -13.180;
   1:L PR[91] 10mm/sec CNT100;
   1:  PR[GP1:91,1] = PR[GP1:90,1] + -44.472;
   1:  PR[GP1:91,2] = PR[GP1:90,2] + -23.428;
   1:L PR[91] 10mm/sec CNT100;
   1:  PR[GP1:91,1] = PR[GP1:90,1] + -43.336;
   1:  PR[GP1:91,2] = PR[GP1:90,2] + -25.522;
   1:L PR[91] 10mm/sec CNT100;
   1:  PR[GP1:91,1] = PR[GP1:90,1] + -36.138;
   1:  PR[GP1:91,2] = PR[GP1:90,2] + -34.192;
   1:L PR[91] 10mm/sec CNT100;
   1:  PR[GP1:91,1] = PR[GP1:90,1] + -34.437;
   1:  PR[GP1:91,2] = PR[GP1:90,2] + -35.771;
   1:L PR[91] 10mm/sec CNT100;
   1:  PR[GP1:91,1] = PR[GP1:90,1] + -21.572;
   1:  PR[GP1:91,2] = PR[GP1:90,2] + -43.739;
   1:L PR[91] 10mm/sec CNT100;
   1:  PR[GP1:91,1] = PR[GP1:90,1] + -19.516;
   1:  PR[GP1:91,2] = PR[GP1:90,2] + -44.679;
   1:L PR[91] 10mm/sec CNT100;
   1:  PR[GP1:91,1] = PR[GP1:90,1] + -4.518;
   1:  PR[GP1:91,2] = PR[GP1:90,2] + -47.484;
   1:L PR[91] 10mm/sec CNT100;
   1:  PR[GP1:91,1] = PR[GP1:90,1] + -2.335;
   1:  PR[GP1:91,2] = PR[GP1:90,2] + -47.724;
   1:L PR[91] 10mm/sec CNT100;
   1:  PR[GP1:91,1] = PR[GP1:90,1] + -0.265;
   1:  PR[GP1:91,2] = PR[GP1:90,2] + -47.377;
   1:L PR[91] 10mm/sec CNT100;
   1:  PR[GP1:91,1] = PR[GP1:90,1] + 1.612;
   1:  PR[GP1:91,2] = PR[GP1:90,2] + -47.852;
   1:  PR[GP1:91,3] = PR[GP1:90,3] + 122.305;
   1:L PR[91] 10mm/sec CNT100;
   1:  PR[GP1:91,1] = PR[GP1:90,1] + 3.584;
   1:  PR[GP1:91,2] = PR[GP1:90,2] + -47.635;
   1:L PR[91] 10mm/sec CNT100;
   1:  PR[GP1:91,1] = PR[GP1:90,1] + 18.860;
   1:  PR[GP1:91,2] = PR[GP1:90,2] + -44.780;
   1:L PR[91] 10mm/sec CNT100;
   1:  PR[GP1:91,1] = PR[GP1:90,1] + 20.718;
   1:  PR[GP1:91,2] = PR[GP1:90,2] + -43.932;
   1:L PR[91] 10mm/sec CNT100;
   1:  PR[GP1:91,1] = PR[GP1:90,1] + 33.834;
   1:  PR[GP1:91,2] = PR[GP1:90,2] + -35.809;
   1:L PR[91] 10mm/sec CNT100;
   1:  PR[GP1:91,1] = PR[GP1:90,1] + 35.371;
   1:  PR[GP1:91,2] = PR[GP1:90,2] + -34.380;
   1:L PR[91] 10mm/sec CNT100;
   1:  PR[GP1:91,1] = PR[GP1:90,1] + 42.712;
   1:  PR[GP1:91,2] = PR[GP1:90,2] + -25.537;
   1:L PR[91] 10mm/sec CNT100;
   1:  PR[GP1:91,1] = PR[GP1:90,1] + 43.740;
   1:  PR[GP1:91,2] = PR[GP1:90,2] + -23.646;
   1:L PR[91] 10mm/sec CNT100;
   1:  PR[GP1:91,1] = PR[GP1:90,1] + 48.361;
   1:  PR[GP1:91,2] = PR[GP1:90,2] + -13.179;
   1:L PR[91] 10mm/sec CNT100;
   1:  PR[GP1:91,1] = PR[GP1:90,1] + 48.720;
   1:  PR[GP1:91,2] = PR[GP1:90,2] + -11.042;
   1:L PR[91] 10mm/sec CNT100;
   1:  PR[GP1:91,1] = PR[GP1:90,1] + 50.291;
   1:  PR[GP1:91,2] = PR[GP1:90,2] + 0.271;
   1:L PR[91] 10mm/sec CNT100;
   1:  PR[GP1:91,1] = PR[GP1:90,1] + 49.939;
   1:  PR[GP1:91,2] = PR[GP1:90,2] + 2.393;
   1:L PR[91] 10mm/sec CNT100;
   1:  PR[GP1:91,1] = PR[GP1:90,1] + 48.356;
   1:  PR[GP1:91,2] = PR[GP1:90,2] + 13.749;
   1:L PR[91] 10mm/sec CNT100;
   1:  PR[GP1:91,1] = PR[GP1:90,1] + 43.738;
   1:  PR[GP1:91,2] = PR[GP1:90,2] + 24.208;
   1:L PR[91] 10mm/sec CNT100;
   1:  PR[GP1:91,1] = PR[GP1:90,1] + 42.707;
   1:  PR[GP1:91,2] = PR[GP1:90,2] + 26.102;
   1:L PR[91] 10mm/sec CNT100;
   1:  PR[GP1:91,1] = PR[GP1:90,1] + 35.366;
   1:  PR[GP1:91,2] = PR[GP1:90,2] + 34.945;
   1:L PR[91] 10mm/sec CNT100;
   1:  PR[GP1:91,1] = PR[GP1:90,1] + 33.823;
   1:  PR[GP1:91,2] = PR[GP1:90,2] + 36.374;
   1:L PR[91] 10mm/sec CNT100;
   1:  PR[GP1:91,1] = PR[GP1:90,1] + 20.706;
   1:  PR[GP1:91,2] = PR[GP1:90,2] + 44.498;
   1:L PR[91] 10mm/sec CNT100;
   1:  PR[GP1:91,1] = PR[GP1:90,1] + 18.844;
   1:  PR[GP1:91,2] = PR[GP1:90,2] + 45.343;
   1:L PR[91] 10mm/sec CNT100;
   1:  PR[GP1:91,1] = PR[GP1:90,1] + 3.567;
   1:  PR[GP1:91,2] = PR[GP1:90,2] + 48.198;
   1:L PR[91] 10mm/sec CNT100;
   1:  PR[GP1:91,1] = PR[GP1:90,1] + 1.594;
   1:  PR[GP1:91,2] = PR[GP1:90,2] + 48.409;
   1:L PR[91] 10mm/sec CNT100;
   1:  PR[GP1:91,1] = PR[GP1:90,1] + -0.266;
   1:  PR[GP1:91,2] = PR[GP1:90,2] + 48.082;
   1:L PR[91] 10mm/sec CNT100;
   1:  PR[GP1:91,1] = PR[GP1:90,1] + -2.127;
   1:  PR[GP1:91,2] = PR[GP1:90,2] + 48.409;
   1:L PR[91] 10mm/sec CNT100;
   1:  PR[GP1:91,1] = PR[GP1:90,1] + -4.100;
   1:  PR[GP1:91,2] = PR[GP1:90,2] + 48.198;
   1:L PR[91] 10mm/sec CNT100;
   1:  PR[GP1:91,1] = PR[GP1:90,1] + -19.373;
   1:  PR[GP1:91,2] = PR[GP1:90,2] + 45.342;
   1:L PR[91] 10mm/sec CNT100;
   1:  PR[GP1:91,1] = PR[GP1:90,1] + -21.235;
   1:  PR[GP1:91,2] = PR[GP1:90,2] + 44.496;
   1:L PR[91] 10mm/sec CNT100;
   1:  PR[GP1:91,1] = PR[GP1:90,1] + -34.348;
   1:  PR[GP1:91,2] = PR[GP1:90,2] + 36.375;
   1:L PR[91] 10mm/sec CNT100;
   1:  PR[GP1:91,1] = PR[GP1:90,1] + -35.891;
   1:  PR[GP1:91,2] = PR[GP1:90,2] + 34.947;
   1:L PR[91] 10mm/sec CNT100;
   1:  PR[GP1:91,1] = PR[GP1:90,1] + -43.232;
   1:  PR[GP1:91,2] = PR[GP1:90,2] + 26.104;
   1:L PR[91] 10mm/sec CNT100;
   1:  PR[GP1:91,1] = PR[GP1:90,1] + -44.264;
   1:  PR[GP1:91,2] = PR[GP1:90,2] + 24.207;
   1:L PR[91] 10mm/sec CNT100;
   1:  PR[GP1:91,1] = PR[GP1:90,1] + -48.885;
   1:  PR[GP1:91,2] = PR[GP1:90,2] + 13.741;
   1:L PR[91] 10mm/sec CNT100;
   1:  PR[GP1:91,1] = PR[GP1:90,1] + -49.246;
   1:  PR[GP1:91,2] = PR[GP1:90,2] + 11.546;
   1:L PR[91] 10mm/sec CNT100;
   1:  PR[GP1:91,1] = PR[GP1:90,1] + -50.817;
   1:  PR[GP1:91,2] = PR[GP1:90,2] + 0.287;
   1:L PR[91] 10mm/sec CNT100;
   1:  PR[GP1:91,1] = PR[GP1:90,1] + -50.467;
   1:  PR[GP1:91,2] = PR[GP1:90,2] + -1.828;
   1:L PR[91] 10mm/sec CNT100;
   1:  PR[GP1:91,1] = PR[GP1:90,1] + -48.883;
   1:  PR[GP1:91,2] = PR[GP1:90,2] + -13.185;
   1:L PR[91] 10mm/sec CNT100;
   1:  PR[GP1:91,1] = PR[GP1:90,1] + -44.266;
   1:  PR[GP1:91,2] = PR[GP1:90,2] + -23.644;
   1:L PR[91] 10mm/sec CNT100;
   1:  PR[GP1:91,1] = PR[GP1:90,1] + -43.238;
   1:  PR[GP1:91,2] = PR[GP1:90,2] + -25.539;
   1:L PR[91] 10mm/sec CNT100;
   1:  PR[GP1:91,1] = PR[GP1:90,1] + -35.896;
   1:  PR[GP1:91,2] = PR[GP1:90,2] + -34.382;
   1:L PR[91] 10mm/sec CNT100;
   1:  PR[GP1:91,1] = PR[GP1:90,1] + -34.359;
   1:  PR[GP1:91,2] = PR[GP1:90,2] + -35.810;
   1:L PR[91] 10mm/sec CNT100;
   1:  PR[GP1:91,1] = PR[GP1:90,1] + -21.247;
   1:  PR[GP1:91,2] = PR[GP1:90,2] + -43.931;
   1:L PR[91] 10mm/sec CNT100;
   1:  PR[GP1:91,1] = PR[GP1:90,1] + -19.389;
   1:  PR[GP1:91,2] = PR[GP1:90,2] + -44.779;
   1:L PR[91] 10mm/sec CNT100;
   1:  PR[GP1:91,1] = PR[GP1:90,1] + -4.117;
   1:  PR[GP1:91,2] = PR[GP1:90,2] + -47.636;
   1:L PR[91] 10mm/sec CNT100;
   1:  PR[GP1:91,1] = PR[GP1:90,1] + -2.146;
   1:  PR[GP1:91,2] = PR[GP1:90,2] + -47.852;
   1:L PR[91] 10mm/sec CNT100;
   1:  PR[GP1:91,1] = PR[GP1:90,1] + -0.266;
   1:  PR[GP1:91,2] = PR[GP1:90,2] + -47.537;
   1:L PR[91] 10mm/sec CNT100;
   1:  PR[GP1:91,1] = PR[GP1:90,1] + 1.423;
   1:  PR[GP1:91,2] = PR[GP1:90,2] + -47.980;
   1:  PR[GP1:91,3] = PR[GP1:90,3] + 122.915;
   1:L PR[91] 10mm/sec CNT100;
   1:  PR[GP1:91,1] = PR[GP1:90,1] + 3.183;
   1:  PR[GP1:91,2] = PR[GP1:90,2] + -47.787;
   1:L PR[91] 10mm/sec CNT100;
   1:  PR[GP1:91,1] = PR[GP1:90,1] + 18.734;
   1:  PR[GP1:91,2] = PR[GP1:90,2] + -44.880;
   1:L PR[91] 10mm/sec CNT100;
   1:  PR[GP1:91,1] = PR[GP1:90,1] + 20.392;
   1:  PR[GP1:91,2] = PR[GP1:90,2] + -44.123;
   1:L PR[91] 10mm/sec CNT100;
